Fanuc TP program (LS listing): layer_407.ls

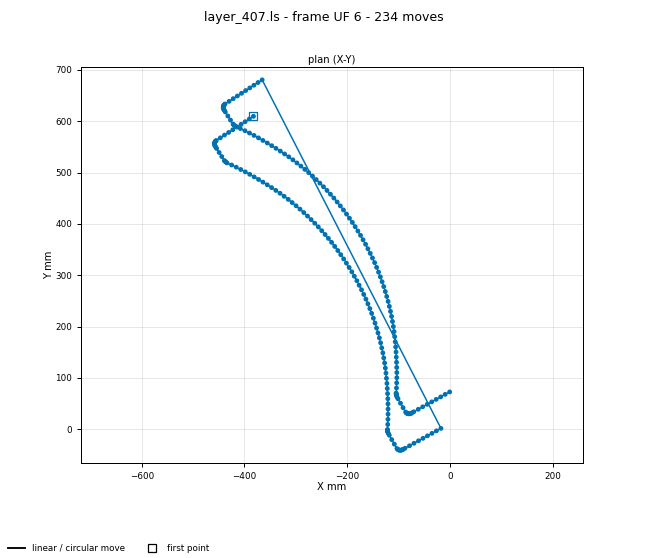
[picture p0: tool path of layer_407.ls in frame UF 6, 234 of 234 moves have a stored position in this frame; points joined in program order, loops and branches not executed]
/PROG layer_407
/ATTR
OWNER       = MNEDITOR;
CREATE      = DATE 100-11-20  TIME 09:43:21;
MODIFIED    = DATE 100-12-05  TIME 05:26:29;
LINE_COUNT = 119;
PROTECT     = READ_WRITE;
TCD:  STACK_SIZE    = 0,
      TASK_PRIORITY = 50,
      TIME_SLICE    = 0,
      BUSY_LAMP_OFF = 0,
      ABORT_REQUEST = 0,
      PAUSE_REQUEST = 0;
DEFAULT_GROUP   = 1,1,*,*,*;
CONTROL_CODE    = 00000000 00000000;
/MN
:R[35]=920.0;
:R[34]=0;
1: L P[1] 240cm/min CNT100 COORD ;
: Arc Start[1];
2: L P[2] 240cm/min CNT100 COORD PTH ;
3: L P[3] 240cm/min CNT100 COORD PTH ;
4: L P[4] 240cm/min CNT100 COORD PTH ;
5: L P[5] 240cm/min CNT100 COORD PTH ;
6: L P[6] 240cm/min CNT100 COORD PTH ;
7: L P[7] 240cm/min CNT100 COORD PTH ;
8: L P[8] 240cm/min CNT100 COORD PTH ;
9: L P[9] 240cm/min CNT100 COORD PTH ;
10: L P[10] 240cm/min CNT100 COORD PTH ;
11: L P[11] 240cm/min CNT100 COORD PTH ;
12: L P[12] 240cm/min CNT100 COORD PTH ;
13: L P[13] 240cm/min CNT100 COORD PTH ;
14: L P[14] 240cm/min CNT100 COORD PTH ;
15: L P[15] 240cm/min CNT100 COORD PTH ;
16: L P[16] 240cm/min CNT100 COORD PTH ;
17: L P[17] 240cm/min CNT100 COORD PTH ;
18: L P[18] 240cm/min CNT100 COORD PTH ;
19: L P[19] 240cm/min CNT100 COORD PTH ;
20: L P[20] 240cm/min CNT100 COORD PTH ;
21: L P[21] 240cm/min CNT100 COORD PTH ;
22: L P[22] 240cm/min CNT100 COORD PTH ;
23: L P[23] 240cm/min CNT100 COORD PTH ;
24: L P[24] 240cm/min CNT100 COORD PTH ;
25: L P[25] 240cm/min CNT100 COORD PTH ;
26: L P[26] 240cm/min CNT100 COORD PTH ;
27: L P[27] 240cm/min CNT100 COORD PTH ;
28: L P[28] 240cm/min CNT100 COORD PTH ;
29: L P[29] 240cm/min CNT100 COORD PTH ;
30: L P[30] 240cm/min CNT100 COORD PTH ;
31: L P[31] 240cm/min CNT100 COORD PTH ;
32: L P[32] 240cm/min CNT100 COORD PTH ;
33: L P[33] 240cm/min CNT100 COORD PTH ;
34: L P[34] 240cm/min CNT100 COORD PTH ;
35: L P[35] 240cm/min CNT100 COORD PTH ;
36: L P[36] 240cm/min CNT100 COORD PTH ;
37: L P[37] 240cm/min CNT100 COORD PTH ;
38: L P[38] 240cm/min CNT100 COORD PTH ;
39: L P[39] 240cm/min CNT100 COORD PTH ;
40: L P[40] 240cm/min CNT100 COORD PTH ;
41: L P[41] 240cm/min CNT100 COORD PTH ;
42: L P[42] 240cm/min CNT100 COORD PTH ;
43: L P[43] 240cm/min CNT100 COORD PTH ;
44: L P[44] 240cm/min CNT100 COORD PTH ;
45: L P[45] 240cm/min CNT100 COORD PTH ;
46: L P[46] 240cm/min CNT100 COORD PTH ;
47: L P[47] 240cm/min CNT100 COORD PTH ;
48: L P[48] 240cm/min CNT100 COORD PTH ;
49: L P[49] 240cm/min CNT100 COORD PTH ;
50: L P[50] 240cm/min CNT100 COORD PTH ;
51: L P[51] 240cm/min CNT100 COORD PTH ;
52: L P[52] 240cm/min CNT100 COORD PTH ;
53: L P[53] 240cm/min CNT100 COORD PTH ;
54: L P[54] 240cm/min CNT100 COORD PTH ;
55: L P[55] 240cm/min CNT100 COORD PTH ;
56: L P[56] 240cm/min CNT100 COORD PTH ;
57: L P[57] 240cm/min CNT100 COORD PTH ;
58: L P[58] 240cm/min CNT100 COORD PTH ;
59: L P[59] 240cm/min CNT100 COORD PTH ;
60: L P[60] 240cm/min CNT100 COORD PTH ;
61: L P[61] 240cm/min CNT100 COORD PTH ;
62: L P[62] 240cm/min CNT100 COORD PTH ;
63: L P[63] 240cm/min CNT100 COORD PTH ;
64: L P[64] 240cm/min CNT100 COORD PTH ;
65: L P[65] 240cm/min CNT100 COORD PTH ;
66: L P[66] 240cm/min CNT100 COORD PTH ;
67: L P[67] 240cm/min CNT100 COORD PTH ;
68: L P[68] 240cm/min CNT100 COORD PTH ;
69: L P[69] 240cm/min CNT100 COORD PTH ;
70: L P[70] 240cm/min CNT100 COORD PTH ;
71: L P[71] 240cm/min CNT100 COORD PTH ;
72: L P[72] 240cm/min CNT100 COORD PTH ;
73: L P[73] 240cm/min CNT100 COORD PTH ;
74: L P[74] 240cm/min CNT100 COORD PTH ;
75: L P[75] 240cm/min CNT100 COORD PTH ;
76: L P[76] 240cm/min CNT100 COORD PTH ;
77: L P[77] 240cm/min CNT100 COORD PTH ;
78: L P[78] 240cm/min CNT100 COORD PTH ;
79: L P[79] 240cm/min CNT100 COORD PTH ;
80: L P[80] 240cm/min CNT100 COORD PTH ;
81: L P[81] 240cm/min CNT100 COORD PTH ;
82: L P[82] 240cm/min CNT100 COORD PTH ;
83: L P[83] 240cm/min CNT100 COORD PTH ;
84: L P[84] 240cm/min CNT100 COORD PTH ;
85: L P[85] 240cm/min CNT100 COORD PTH ;
86: L P[86] 240cm/min CNT100 COORD PTH ;
87: L P[87] 240cm/min CNT100 COORD PTH ;
88: L P[88] 240cm/min CNT100 COORD PTH ;
89: L P[89] 240cm/min CNT100 COORD PTH ;
90: L P[90] 240cm/min CNT100 COORD PTH ;
91: L P[91] 240cm/min CNT100 COORD PTH ;
92: L P[92] 240cm/min CNT100 COORD PTH ;
93: L P[93] 240cm/min CNT100 COORD PTH ;
94: L P[94] 240cm/min CNT100 COORD PTH ;
95: L P[95] 240cm/min CNT100 COORD PTH ;
96: L P[96] 240cm/min CNT100 COORD PTH ;
97: L P[97] 240cm/min CNT100 COORD PTH ;
98: L P[98] 240cm/min CNT100 COORD PTH ;
99: L P[99] 240cm/min CNT100 COORD PTH ;
100: L P[100] 240cm/min CNT100 COORD PTH ;
101: L P[101] 240cm/min CNT100 COORD PTH ;
102: L P[102] 240cm/min CNT100 COORD PTH ;
103: L P[103] 240cm/min CNT100 COORD PTH ;
104: L P[104] 240cm/min CNT100 COORD PTH ;
105: L P[105] 240cm/min CNT100 COORD PTH ;
106: L P[106] 240cm/min CNT100 COORD PTH ;
107: L P[107] 240cm/min CNT100 COORD PTH ;
108: L P[108] 240cm/min CNT100 COORD PTH ;
109: L P[109] 240cm/min CNT100 COORD PTH ;
110: L P[110] 240cm/min CNT100 COORD PTH ;
111: L P[111] 240cm/min CNT100 COORD PTH ;
112: L P[112] 240cm/min CNT100 COORD PTH ;
113: L P[113] 240cm/min CNT100 COORD PTH ;
114: L P[114] 240cm/min CNT100 COORD PTH ;
115: L P[115] 240cm/min CNT100 COORD PTH ;
116: L P[116] 240cm/min CNT100 COORD PTH ;
117: L P[117] 240cm/min CNT100 COORD PTH ;
: Arc End[1];
:R[34]=1;
:SR[23]=$SCR_GRP[1].$MCH_POS_X;
:SR[24]=$SCR_GRP[1].$MCH_POS_Y;
120: L P[120] 800cm/min CNT100 COORD ;
:SR[23]=$SCR_GRP[1].$MCH_POS_X;
:SR[24]=$SCR_GRP[1].$MCH_POS_Y;
121: L P[121] 800cm/min CNT100 COORD PTH ;
:SR[23]=$SCR_GRP[1].$MCH_POS_X;
:SR[24]=$SCR_GRP[1].$MCH_POS_Y;
122: L P[122] 800cm/min CNT100 COORD PTH ;
:SR[23]=$SCR_GRP[1].$MCH_POS_X;
:SR[24]=$SCR_GRP[1].$MCH_POS_Y;
123: L P[123] 800cm/min CNT100 COORD PTH ;
:SR[23]=$SCR_GRP[1].$MCH_POS_X;
:SR[24]=$SCR_GRP[1].$MCH_POS_Y;
124: L P[124] 800cm/min CNT100 COORD PTH ;
:SR[23]=$SCR_GRP[1].$MCH_POS_X;
:SR[24]=$SCR_GRP[1].$MCH_POS_Y;
125: L P[125] 800cm/min CNT100 COORD PTH ;
:SR[23]=$SCR_GRP[1].$MCH_POS_X;
:SR[24]=$SCR_GRP[1].$MCH_POS_Y;
126: L P[126] 800cm/min CNT100 COORD PTH ;
:SR[23]=$SCR_GRP[1].$MCH_POS_X;
:SR[24]=$SCR_GRP[1].$MCH_POS_Y;
127: L P[127] 800cm/min CNT100 COORD PTH ;
:SR[23]=$SCR_GRP[1].$MCH_POS_X;
:SR[24]=$SCR_GRP[1].$MCH_POS_Y;
128: L P[128] 800cm/min CNT100 COORD PTH ;
:SR[23]=$SCR_GRP[1].$MCH_POS_X;
:SR[24]=$SCR_GRP[1].$MCH_POS_Y;
129: L P[129] 800cm/min CNT100 COORD PTH ;
:SR[23]=$SCR_GRP[1].$MCH_POS_X;
:SR[24]=$SCR_GRP[1].$MCH_POS_Y;
130: L P[130] 800cm/min CNT100 COORD PTH ;
:SR[23]=$SCR_GRP[1].$MCH_POS_X;
:SR[24]=$SCR_GRP[1].$MCH_POS_Y;
131: L P[131] 800cm/min CNT100 COORD PTH ;
:SR[23]=$SCR_GRP[1].$MCH_POS_X;
:SR[24]=$SCR_GRP[1].$MCH_POS_Y;
132: L P[132] 800cm/min CNT100 COORD PTH ;
:SR[23]=$SCR_GRP[1].$MCH_POS_X;
:SR[24]=$SCR_GRP[1].$MCH_POS_Y;
133: L P[133] 800cm/min CNT100 COORD PTH ;
:SR[23]=$SCR_GRP[1].$MCH_POS_X;
:SR[24]=$SCR_GRP[1].$MCH_POS_Y;
134: L P[134] 800cm/min CNT100 COORD PTH ;
:SR[23]=$SCR_GRP[1].$MCH_POS_X;
:SR[24]=$SCR_GRP[1].$MCH_POS_Y;
135: L P[135] 800cm/min CNT100 COORD PTH ;
:SR[23]=$SCR_GRP[1].$MCH_POS_X;
:SR[24]=$SCR_GRP[1].$MCH_POS_Y;
136: L P[136] 800cm/min CNT100 COORD PTH ;
:SR[23]=$SCR_GRP[1].$MCH_POS_X;
:SR[24]=$SCR_GRP[1].$MCH_POS_Y;
137: L P[137] 800cm/min CNT100 COORD PTH ;
:SR[23]=$SCR_GRP[1].$MCH_POS_X;
:SR[24]=$SCR_GRP[1].$MCH_POS_Y;
138: L P[138] 800cm/min CNT100 COORD PTH ;
:SR[23]=$SCR_GRP[1].$MCH_POS_X;
:SR[24]=$SCR_GRP[1].$MCH_POS_Y;
139: L P[139] 800cm/min CNT100 COORD PTH ;
:SR[23]=$SCR_GRP[1].$MCH_POS_X;
:SR[24]=$SCR_GRP[1].$MCH_POS_Y;
140: L P[140] 800cm/min CNT100 COORD PTH ;
:SR[23]=$SCR_GRP[1].$MCH_POS_X;
:SR[24]=$SCR_GRP[1].$MCH_POS_Y;
141: L P[141] 800cm/min CNT100 COORD PTH ;
:SR[23]=$SCR_GRP[1].$MCH_POS_X;
:SR[24]=$SCR_GRP[1].$MCH_POS_Y;
142: L P[142] 800cm/min CNT100 COORD PTH ;
:SR[23]=$SCR_GRP[1].$MCH_POS_X;
:SR[24]=$SCR_GRP[1].$MCH_POS_Y;
143: L P[143] 800cm/min CNT100 COORD PTH ;
:SR[23]=$SCR_GRP[1].$MCH_POS_X;
:SR[24]=$SCR_GRP[1].$MCH_POS_Y;
144: L P[144] 800cm/min CNT100 COORD PTH ;
:SR[23]=$SCR_GRP[1].$MCH_POS_X;
:SR[24]=$SCR_GRP[1].$MCH_POS_Y;
145: L P[145] 800cm/min CNT100 COORD PTH ;
:SR[23]=$SCR_GRP[1].$MCH_POS_X;
:SR[24]=$SCR_GRP[1].$MCH_POS_Y;
146: L P[146] 800cm/min CNT100 COORD PTH ;
:SR[23]=$SCR_GRP[1].$MCH_POS_X;
:SR[24]=$SCR_GRP[1].$MCH_POS_Y;
147: L P[147] 800cm/min CNT100 COORD PTH ;
:SR[23]=$SCR_GRP[1].$MCH_POS_X;
:SR[24]=$SCR_GRP[1].$MCH_POS_Y;
148: L P[148] 800cm/min CNT100 COORD PTH ;
:SR[23]=$SCR_GRP[1].$MCH_POS_X;
:SR[24]=$SCR_GRP[1].$MCH_POS_Y;
149: L P[149] 800cm/min CNT100 COORD PTH ;
:SR[23]=$SCR_GRP[1].$MCH_POS_X;
:SR[24]=$SCR_GRP[1].$MCH_POS_Y;
150: L P[150] 800cm/min CNT100 COORD PTH ;
:SR[23]=$SCR_GRP[1].$MCH_POS_X;
:SR[24]=$SCR_GRP[1].$MCH_POS_Y;
151: L P[151] 800cm/min CNT100 COORD PTH ;
:SR[23]=$SCR_GRP[1].$MCH_POS_X;
:SR[24]=$SCR_GRP[1].$MCH_POS_Y;
152: L P[152] 800cm/min CNT100 COORD PTH ;
:SR[23]=$SCR_GRP[1].$MCH_POS_X;
:SR[24]=$SCR_GRP[1].$MCH_POS_Y;
153: L P[153] 800cm/min CNT100 COORD PTH ;
:SR[23]=$SCR_GRP[1].$MCH_POS_X;
:SR[24]=$SCR_GRP[1].$MCH_POS_Y;
154: L P[154] 800cm/min CNT100 COORD PTH ;
:SR[23]=$SCR_GRP[1].$MCH_POS_X;
:SR[24]=$SCR_GRP[1].$MCH_POS_Y;
155: L P[155] 800cm/min CNT100 COORD PTH ;
:SR[23]=$SCR_GRP[1].$MCH_POS_X;
:SR[24]=$SCR_GRP[1].$MCH_POS_Y;
156: L P[156] 800cm/min CNT100 COORD PTH ;
:SR[23]=$SCR_GRP[1].$MCH_POS_X;
:SR[24]=$SCR_GRP[1].$MCH_POS_Y;
157: L P[157] 800cm/min CNT100 COORD PTH ;
:SR[23]=$SCR_GRP[1].$MCH_POS_X;
:SR[24]=$SCR_GRP[1].$MCH_POS_Y;
158: L P[158] 800cm/min CNT100 COORD PTH ;
:SR[23]=$SCR_GRP[1].$MCH_POS_X;
:SR[24]=$SCR_GRP[1].$MCH_POS_Y;
159: L P[159] 800cm/min CNT100 COORD PTH ;
:SR[23]=$SCR_GRP[1].$MCH_POS_X;
:SR[24]=$SCR_GRP[1].$MCH_POS_Y;
160: L P[160] 800cm/min CNT100 COORD PTH ;
:SR[23]=$SCR_GRP[1].$MCH_POS_X;
:SR[24]=$SCR_GRP[1].$MCH_POS_Y;
161: L P[161] 800cm/min CNT100 COORD PTH ;
:SR[23]=$SCR_GRP[1].$MCH_POS_X;
:SR[24]=$SCR_GRP[1].$MCH_POS_Y;
162: L P[162] 800cm/min CNT100 COORD PTH ;
:SR[23]=$SCR_GRP[1].$MCH_POS_X;
:SR[24]=$SCR_GRP[1].$MCH_POS_Y;
163: L P[163] 800cm/min CNT100 COORD PTH ;
:SR[23]=$SCR_GRP[1].$MCH_POS_X;
:SR[24]=$SCR_GRP[1].$MCH_POS_Y;
164: L P[164] 800cm/min CNT100 COORD PTH ;
:SR[23]=$SCR_GRP[1].$MCH_POS_X;
:SR[24]=$SCR_GRP[1].$MCH_POS_Y;
165: L P[165] 800cm/min CNT100 COORD PTH ;
:SR[23]=$SCR_GRP[1].$MCH_POS_X;
:SR[24]=$SCR_GRP[1].$MCH_POS_Y;
166: L P[166] 800cm/min CNT100 COORD PTH ;
:SR[23]=$SCR_GRP[1].$MCH_POS_X;
:SR[24]=$SCR_GRP[1].$MCH_POS_Y;
167: L P[167] 800cm/min CNT100 COORD PTH ;
:SR[23]=$SCR_GRP[1].$MCH_POS_X;
:SR[24]=$SCR_GRP[1].$MCH_POS_Y;
168: L P[168] 800cm/min CNT100 COORD PTH ;
:SR[23]=$SCR_GRP[1].$MCH_POS_X;
:SR[24]=$SCR_GRP[1].$MCH_POS_Y;
169: L P[169] 800cm/min CNT100 COORD PTH ;
:SR[23]=$SCR_GRP[1].$MCH_POS_X;
:SR[24]=$SCR_GRP[1].$MCH_POS_Y;
170: L P[170] 800cm/min CNT100 COORD PTH ;
:SR[23]=$SCR_GRP[1].$MCH_POS_X;
:SR[24]=$SCR_GRP[1].$MCH_POS_Y;
171: L P[171] 800cm/min CNT100 COORD PTH ;
:SR[23]=$SCR_GRP[1].$MCH_POS_X;
:SR[24]=$SCR_GRP[1].$MCH_POS_Y;
172: L P[172] 800cm/min CNT100 COORD PTH ;
:SR[23]=$SCR_GRP[1].$MCH_POS_X;
:SR[24]=$SCR_GRP[1].$MCH_POS_Y;
173: L P[173] 800cm/min CNT100 COORD PTH ;
:SR[23]=$SCR_GRP[1].$MCH_POS_X;
:SR[24]=$SCR_GRP[1].$MCH_POS_Y;
174: L P[174] 800cm/min CNT100 COORD PTH ;
:SR[23]=$SCR_GRP[1].$MCH_POS_X;
:SR[24]=$SCR_GRP[1].$MCH_POS_Y;
175: L P[175] 800cm/min CNT100 COORD PTH ;
:SR[23]=$SCR_GRP[1].$MCH_POS_X;
:SR[24]=$SCR_GRP[1].$MCH_POS_Y;
176: L P[176] 800cm/min CNT100 COORD PTH ;
:SR[23]=$SCR_GRP[1].$MCH_POS_X;
:SR[24]=$SCR_GRP[1].$MCH_POS_Y;
177: L P[177] 800cm/min CNT100 COORD PTH ;
:SR[23]=$SCR_GRP[1].$MCH_POS_X;
:SR[24]=$SCR_GRP[1].$MCH_POS_Y;
178: L P[178] 800cm/min CNT100 COORD PTH ;
:SR[23]=$SCR_GRP[1].$MCH_POS_X;
:SR[24]=$SCR_GRP[1].$MCH_POS_Y;
179: L P[179] 800cm/min CNT100 COORD PTH ;
:SR[23]=$SCR_GRP[1].$MCH_POS_X;
:SR[24]=$SCR_GRP[1].$MCH_POS_Y;
180: L P[180] 800cm/min CNT100 COORD PTH ;
:SR[23]=$SCR_GRP[1].$MCH_POS_X;
:SR[24]=$SCR_GRP[1].$MCH_POS_Y;
181: L P[181] 800cm/min CNT100 COORD PTH ;
:SR[23]=$SCR_GRP[1].$MCH_POS_X;
:SR[24]=$SCR_GRP[1].$MCH_POS_Y;
182: L P[182] 800cm/min CNT100 COORD PTH ;
:SR[23]=$SCR_GRP[1].$MCH_POS_X;
:SR[24]=$SCR_GRP[1].$MCH_POS_Y;
183: L P[183] 800cm/min CNT100 COORD PTH ;
:SR[23]=$SCR_GRP[1].$MCH_POS_X;
:SR[24]=$SCR_GRP[1].$MCH_POS_Y;
184: L P[184] 800cm/min CNT100 COORD PTH ;
:SR[23]=$SCR_GRP[1].$MCH_POS_X;
:SR[24]=$SCR_GRP[1].$MCH_POS_Y;
185: L P[185] 800cm/min CNT100 COORD PTH ;
:SR[23]=$SCR_GRP[1].$MCH_POS_X;
:SR[24]=$SCR_GRP[1].$MCH_POS_Y;
186: L P[186] 800cm/min CNT100 COORD PTH ;
:SR[23]=$SCR_GRP[1].$MCH_POS_X;
:SR[24]=$SCR_GRP[1].$MCH_POS_Y;
187: L P[187] 800cm/min CNT100 COORD PTH ;
:SR[23]=$SCR_GRP[1].$MCH_POS_X;
:SR[24]=$SCR_GRP[1].$MCH_POS_Y;
188: L P[188] 800cm/min CNT100 COORD PTH ;
:SR[23]=$SCR_GRP[1].$MCH_POS_X;
:SR[24]=$SCR_GRP[1].$MCH_POS_Y;
189: L P[189] 800cm/min CNT100 COORD PTH ;
:SR[23]=$SCR_GRP[1].$MCH_POS_X;
:SR[24]=$SCR_GRP[1].$MCH_POS_Y;
190: L P[190] 800cm/min CNT100 COORD PTH ;
:SR[23]=$SCR_GRP[1].$MCH_POS_X;
:SR[24]=$SCR_GRP[1].$MCH_POS_Y;
191: L P[191] 800cm/min CNT100 COORD PTH ;
:SR[23]=$SCR_GRP[1].$MCH_POS_X;
:SR[24]=$SCR_GRP[1].$MCH_POS_Y;
192: L P[192] 800cm/min CNT100 COORD PTH ;
:SR[23]=$SCR_GRP[1].$MCH_POS_X;
:SR[24]=$SCR_GRP[1].$MCH_POS_Y;
193: L P[193] 800cm/min CNT100 COORD PTH ;
:SR[23]=$SCR_GRP[1].$MCH_POS_X;
:SR[24]=$SCR_GRP[1].$MCH_POS_Y;
194: L P[194] 800cm/min CNT100 COORD PTH ;
:SR[23]=$SCR_GRP[1].$MCH_POS_X;
:SR[24]=$SCR_GRP[1].$MCH_POS_Y;
195: L P[195] 800cm/min CNT100 COORD PTH ;
:SR[23]=$SCR_GRP[1].$MCH_POS_X;
:SR[24]=$SCR_GRP[1].$MCH_POS_Y;
196: L P[196] 800cm/min CNT100 COORD PTH ;
:SR[23]=$SCR_GRP[1].$MCH_POS_X;
:SR[24]=$SCR_GRP[1].$MCH_POS_Y;
197: L P[197] 800cm/min CNT100 COORD PTH ;
:SR[23]=$SCR_GRP[1].$MCH_POS_X;
:SR[24]=$SCR_GRP[1].$MCH_POS_Y;
198: L P[198] 800cm/min CNT100 COORD PTH ;
:SR[23]=$SCR_GRP[1].$MCH_POS_X;
:SR[24]=$SCR_GRP[1].$MCH_POS_Y;
199: L P[199] 800cm/min CNT100 COORD PTH ;
:SR[23]=$SCR_GRP[1].$MCH_POS_X;
:SR[24]=$SCR_GRP[1].$MCH_POS_Y;
200: L P[200] 800cm/min CNT100 COORD PTH ;
:SR[23]=$SCR_GRP[1].$MCH_POS_X;
:SR[24]=$SCR_GRP[1].$MCH_POS_Y;
201: L P[201] 800cm/min CNT100 COORD PTH ;
:SR[23]=$SCR_GRP[1].$MCH_POS_X;
:SR[24]=$SCR_GRP[1].$MCH_POS_Y;
202: L P[202] 800cm/min CNT100 COORD PTH ;
:SR[23]=$SCR_GRP[1].$MCH_POS_X;
:SR[24]=$SCR_GRP[1].$MCH_POS_Y;
203: L P[203] 800cm/min CNT100 COORD PTH ;
:SR[23]=$SCR_GRP[1].$MCH_POS_X;
:SR[24]=$SCR_GRP[1].$MCH_POS_Y;
204: L P[204] 800cm/min CNT100 COORD PTH ;
:SR[23]=$SCR_GRP[1].$MCH_POS_X;
:SR[24]=$SCR_GRP[1].$MCH_POS_Y;
205: L P[205] 800cm/min CNT100 COORD PTH ;
:SR[23]=$SCR_GRP[1].$MCH_POS_X;
:SR[24]=$SCR_GRP[1].$MCH_POS_Y;
206: L P[206] 800cm/min CNT100 COORD PTH ;
:SR[23]=$SCR_GRP[1].$MCH_POS_X;
:SR[24]=$SCR_GRP[1].$MCH_POS_Y;
207: L P[207] 800cm/min CNT100 COORD PTH ;
:SR[23]=$SCR_GRP[1].$MCH_POS_X;
:SR[24]=$SCR_GRP[1].$MCH_POS_Y;
208: L P[208] 800cm/min CNT100 COORD PTH ;
:SR[23]=$SCR_GRP[1].$MCH_POS_X;
:SR[24]=$SCR_GRP[1].$MCH_POS_Y;
209: L P[209] 800cm/min CNT100 COORD PTH ;
:SR[23]=$SCR_GRP[1].$MCH_POS_X;
:SR[24]=$SCR_GRP[1].$MCH_POS_Y;
210: L P[210] 800cm/min CNT100 COORD PTH ;
:SR[23]=$SCR_GRP[1].$MCH_POS_X;
:SR[24]=$SCR_GRP[1].$MCH_POS_Y;
211: L P[211] 800cm/min CNT100 COORD PTH ;
:SR[23]=$SCR_GRP[1].$MCH_POS_X;
:SR[24]=$SCR_GRP[1].$MCH_POS_Y;
212: L P[212] 800cm/min CNT100 COORD PTH ;
:SR[23]=$SCR_GRP[1].$MCH_POS_X;
:SR[24]=$SCR_GRP[1].$MCH_POS_Y;
213: L P[213] 800cm/min CNT100 COORD PTH ;
:SR[23]=$SCR_GRP[1].$MCH_POS_X;
:SR[24]=$SCR_GRP[1].$MCH_POS_Y;
214: L P[214] 800cm/min CNT100 COORD PTH ;
:SR[23]=$SCR_GRP[1].$MCH_POS_X;
:SR[24]=$SCR_GRP[1].$MCH_POS_Y;
215: L P[215] 800cm/min CNT100 COORD PTH ;
:SR[23]=$SCR_GRP[1].$MCH_POS_X;
:SR[24]=$SCR_GRP[1].$MCH_POS_Y;
216: L P[216] 800cm/min CNT100 COORD PTH ;
:SR[23]=$SCR_GRP[1].$MCH_POS_X;
:SR[24]=$SCR_GRP[1].$MCH_POS_Y;
217: L P[217] 800cm/min CNT100 COORD PTH ;
:SR[23]=$SCR_GRP[1].$MCH_POS_X;
:SR[24]=$SCR_GRP[1].$MCH_POS_Y;
218: L P[218] 800cm/min CNT100 COORD PTH ;
:SR[23]=$SCR_GRP[1].$MCH_POS_X;
:SR[24]=$SCR_GRP[1].$MCH_POS_Y;
219: L P[219] 800cm/min CNT100 COORD PTH ;
:SR[23]=$SCR_GRP[1].$MCH_POS_X;
:SR[24]=$SCR_GRP[1].$MCH_POS_Y;
220: L P[220] 800cm/min CNT100 COORD PTH ;
:SR[23]=$SCR_GRP[1].$MCH_POS_X;
:SR[24]=$SCR_GRP[1].$MCH_POS_Y;
221: L P[221] 800cm/min CNT100 COORD PTH ;
:SR[23]=$SCR_GRP[1].$MCH_POS_X;
:SR[24]=$SCR_GRP[1].$MCH_POS_Y;
222: L P[222] 800cm/min CNT100 COORD PTH ;
:SR[23]=$SCR_GRP[1].$MCH_POS_X;
:SR[24]=$SCR_GRP[1].$MCH_POS_Y;
223: L P[223] 800cm/min CNT100 COORD PTH ;
:SR[23]=$SCR_GRP[1].$MCH_POS_X;
:SR[24]=$SCR_GRP[1].$MCH_POS_Y;
224: L P[224] 800cm/min CNT100 COORD PTH ;
:SR[23]=$SCR_GRP[1].$MCH_POS_X;
:SR[24]=$SCR_GRP[1].$MCH_POS_Y;
225: L P[225] 800cm/min CNT100 COORD PTH ;
:SR[23]=$SCR_GRP[1].$MCH_POS_X;
:SR[24]=$SCR_GRP[1].$MCH_POS_Y;
226: L P[226] 800cm/min CNT100 COORD PTH ;
:SR[23]=$SCR_GRP[1].$MCH_POS_X;
:SR[24]=$SCR_GRP[1].$MCH_POS_Y;
227: L P[227] 800cm/min CNT100 COORD PTH ;
:SR[23]=$SCR_GRP[1].$MCH_POS_X;
:SR[24]=$SCR_GRP[1].$MCH_POS_Y;
228: L P[228] 800cm/min CNT100 COORD PTH ;
:SR[23]=$SCR_GRP[1].$MCH_POS_X;
:SR[24]=$SCR_GRP[1].$MCH_POS_Y;
229: L P[229] 800cm/min CNT100 COORD PTH ;
:SR[23]=$SCR_GRP[1].$MCH_POS_X;
:SR[24]=$SCR_GRP[1].$MCH_POS_Y;
230: L P[230] 800cm/min CNT100 COORD PTH ;
:SR[23]=$SCR_GRP[1].$MCH_POS_X;
:SR[24]=$SCR_GRP[1].$MCH_POS_Y;
231: L P[231] 800cm/min CNT100 COORD PTH ;
:SR[23]=$SCR_GRP[1].$MCH_POS_X;
:SR[24]=$SCR_GRP[1].$MCH_POS_Y;
232: L P[232] 800cm/min CNT100 COORD PTH ;
:SR[23]=$SCR_GRP[1].$MCH_POS_X;
:SR[24]=$SCR_GRP[1].$MCH_POS_Y;
233: L P[233] 800cm/min CNT100 COORD PTH ;
:SR[23]=$SCR_GRP[1].$MCH_POS_X;
:SR[24]=$SCR_GRP[1].$MCH_POS_Y;
234: L P[234] 800cm/min CNT100 COORD PTH ;
:SR[23]=$SCR_GRP[1].$MCH_POS_X;
:SR[24]=$SCR_GRP[1].$MCH_POS_Y;
235: L P[235] 800cm/min CNT100 COORD PTH ;
:SR[23]=$SCR_GRP[1].$MCH_POS_X;
:SR[24]=$SCR_GRP[1].$MCH_POS_Y;
236: L P[236] 800cm/min CNT100 COORD PTH ;
:R[34]=0;
/POS
P[1] {
    GP1:
        UF : 6, UT : 5,     CONFIG: 'N U T, 0, 0, 0',
       X = -382.5 mm, Y = 609.6 mm, Z = 920.0 mm,
       W = 0.0 deg, P = 0.0 deg,
    GP2:
        UF : 1, UT : 2,
       J1 = 0.0 deg, J2 = 0.0 deg
 };
P[120] {
    GP1:
        UF : 6, UT : 5,     CONFIG: 'N U T, 0, 0, 0',
 X = -365.5 mm, Y = 680.6 mm, Z = 920.0 mm,       W = 0.0 deg, P = 0.0 deg,
    GP2:
        UF : 1, UT : 2,
       J1 = 0.0 deg, J2 = 0.0 deg
 };
P[2] {
    GP1:
        UF : 6, UT : 5,     CONFIG: 'N U T, 0, 0, 0',
       X = -390.5 mm, Y = 604.4 mm, Z = 920.0 mm,
       W = 0.0 deg, P = 0.0 deg,
    GP2:
        UF : 1, UT : 2,
       J1 = 0.0 deg, J2 = 0.0 deg
 };
P[121] {
    GP1:
        UF : 6, UT : 5,     CONFIG: 'N U T, 0, 0, 0',
 X = -373.5 mm, Y = 675.4 mm, Z = 920.0 mm,       W = 0.0 deg, P = 0.0 deg,
    GP2:
        UF : 1, UT : 2,
       J1 = 0.0 deg, J2 = 0.0 deg
 };
P[3] {
    GP1:
        UF : 6, UT : 5,     CONFIG: 'N U T, 0, 0, 0',
       X = -398.6 mm, Y = 599.1 mm, Z = 920.0 mm,
       W = 0.0 deg, P = 0.0 deg,
    GP2:
        UF : 1, UT : 2,
       J1 = 0.0 deg, J2 = 0.0 deg
 };
P[122] {
    GP1:
        UF : 6, UT : 5,     CONFIG: 'N U T, 0, 0, 0',
 X = -381.6 mm, Y = 670.1 mm, Z = 920.0 mm,       W = 0.0 deg, P = 0.0 deg,
    GP2:
        UF : 1, UT : 2,
       J1 = 0.0 deg, J2 = 0.0 deg
 };
P[4] {
    GP1:
        UF : 6, UT : 5,     CONFIG: 'N U T, 0, 0, 0',
       X = -406.6 mm, Y = 593.9 mm, Z = 920.0 mm,
       W = 0.0 deg, P = 0.0 deg,
    GP2:
        UF : 1, UT : 2,
       J1 = 0.0 deg, J2 = 0.0 deg
 };
P[123] {
    GP1:
        UF : 6, UT : 5,     CONFIG: 'N U T, 0, 0, 0',
 X = -389.6 mm, Y = 664.9 mm, Z = 920.0 mm,       W = 0.0 deg, P = 0.0 deg,
    GP2:
        UF : 1, UT : 2,
       J1 = 0.0 deg, J2 = 0.0 deg
 };
P[5] {
    GP1:
        UF : 6, UT : 5,     CONFIG: 'N U T, 0, 0, 0',
       X = -414.7 mm, Y = 588.7 mm, Z = 920.0 mm,
       W = 0.0 deg, P = 0.0 deg,
    GP2:
        UF : 1, UT : 2,
       J1 = 0.0 deg, J2 = 0.0 deg
 };
P[124] {
    GP1:
        UF : 6, UT : 5,     CONFIG: 'N U T, 0, 0, 0',
 X = -397.7 mm, Y = 659.7 mm, Z = 920.0 mm,       W = 0.0 deg, P = 0.0 deg,
    GP2:
        UF : 1, UT : 2,
       J1 = 0.0 deg, J2 = 0.0 deg
 };
P[6] {
    GP1:
        UF : 6, UT : 5,     CONFIG: 'N U T, 0, 0, 0',
       X = -422.7 mm, Y = 583.4 mm, Z = 920.0 mm,
       W = 0.0 deg, P = 0.0 deg,
    GP2:
        UF : 1, UT : 2,
       J1 = 0.0 deg, J2 = 0.0 deg
 };
P[125] {
    GP1:
        UF : 6, UT : 5,     CONFIG: 'N U T, 0, 0, 0',
 X = -405.7 mm, Y = 654.4 mm, Z = 920.0 mm,       W = 0.0 deg, P = 0.0 deg,
    GP2:
        UF : 1, UT : 2,
       J1 = 0.0 deg, J2 = 0.0 deg
 };
P[7] {
    GP1:
        UF : 6, UT : 5,     CONFIG: 'N U T, 0, 0, 0',
       X = -430.8 mm, Y = 578.2 mm, Z = 920.0 mm,
       W = 0.0 deg, P = 0.0 deg,
    GP2:
        UF : 1, UT : 2,
       J1 = 0.0 deg, J2 = 0.0 deg
 };
P[126] {
    GP1:
        UF : 6, UT : 5,     CONFIG: 'N U T, 0, 0, 0',
 X = -413.8 mm, Y = 649.2 mm, Z = 920.0 mm,       W = 0.0 deg, P = 0.0 deg,
    GP2:
        UF : 1, UT : 2,
       J1 = 0.0 deg, J2 = 0.0 deg
 };
P[8] {
    GP1:
        UF : 6, UT : 5,     CONFIG: 'N U T, 0, 0, 0',
       X = -438.9 mm, Y = 573.0 mm, Z = 920.0 mm,
       W = 0.0 deg, P = 0.0 deg,
    GP2:
        UF : 1, UT : 2,
       J1 = 0.0 deg, J2 = 0.0 deg
 };
P[127] {
    GP1:
        UF : 6, UT : 5,     CONFIG: 'N U T, 0, 0, 0',
 X = -421.9 mm, Y = 644.0 mm, Z = 920.0 mm,       W = 0.0 deg, P = 0.0 deg,
    GP2:
        UF : 1, UT : 2,
       J1 = 0.0 deg, J2 = 0.0 deg
 };
P[9] {
    GP1:
        UF : 6, UT : 5,     CONFIG: 'N U T, 0, 0, 0',
       X = -446.9 mm, Y = 567.7 mm, Z = 920.0 mm,
       W = 0.0 deg, P = 0.0 deg,
    GP2:
        UF : 1, UT : 2,
       J1 = 0.0 deg, J2 = 0.0 deg
 };
P[128] {
    GP1:
        UF : 6, UT : 5,     CONFIG: 'N U T, 0, 0, 0',
 X = -429.9 mm, Y = 638.7 mm, Z = 920.0 mm,       W = 0.0 deg, P = 0.0 deg,
    GP2:
        UF : 1, UT : 2,
       J1 = 0.0 deg, J2 = 0.0 deg
 };
P[10] {
    GP1:
        UF : 6, UT : 5,     CONFIG: 'N U T, 0, 0, 0',
       X = -455.0 mm, Y = 562.5 mm, Z = 920.0 mm,
       W = 0.0 deg, P = 0.0 deg,
    GP2:
        UF : 1, UT : 2,
       J1 = 0.0 deg, J2 = 0.0 deg
 };
P[129] {
    GP1:
        UF : 6, UT : 5,     CONFIG: 'N U T, 0, 0, 0',
 X = -438.0 mm, Y = 633.5 mm, Z = 920.0 mm,       W = 0.0 deg, P = 0.0 deg,
    GP2:
        UF : 1, UT : 2,
       J1 = 0.0 deg, J2 = 0.0 deg
 };
P[11] {
    GP1:
        UF : 6, UT : 5,     CONFIG: 'N U T, 0, 0, 0',
       X = -456.0 mm, Y = 561.5 mm, Z = 920.0 mm,
       W = 0.0 deg, P = 0.0 deg,
    GP2:
        UF : 1, UT : 2,
       J1 = 0.0 deg, J2 = 0.0 deg
 };
P[130] {
    GP1:
        UF : 6, UT : 5,     CONFIG: 'N U T, 0, 0, 0',
 X = -439.0 mm, Y = 632.5 mm, Z = 920.0 mm,       W = 0.0 deg, P = 0.0 deg,
    GP2:
        UF : 1, UT : 2,
       J1 = 0.0 deg, J2 = 0.0 deg
 };
P[12] {
    GP1:
        UF : 6, UT : 5,     CONFIG: 'N U T, 0, 0, 0',
       X = -456.9 mm, Y = 560.5 mm, Z = 920.0 mm,
       W = 0.0 deg, P = 0.0 deg,
    GP2:
        UF : 1, UT : 2,
       J1 = 0.0 deg, J2 = 0.0 deg
 };
P[131] {
    GP1:
        UF : 6, UT : 5,     CONFIG: 'N U T, 0, 0, 0',
 X = -439.9 mm, Y = 631.5 mm, Z = 920.0 mm,       W = 0.0 deg, P = 0.0 deg,
    GP2:
        UF : 1, UT : 2,
       J1 = 0.0 deg, J2 = 0.0 deg
 };
P[13] {
    GP1:
        UF : 6, UT : 5,     CONFIG: 'N U T, 0, 0, 0',
       X = -457.5 mm, Y = 559.4 mm, Z = 920.0 mm,
       W = 0.0 deg, P = 0.0 deg,
    GP2:
        UF : 1, UT : 2,
       J1 = 0.0 deg, J2 = 0.0 deg
 };
P[132] {
    GP1:
        UF : 6, UT : 5,     CONFIG: 'N U T, 0, 0, 0',
 X = -440.5 mm, Y = 630.4 mm, Z = 920.0 mm,       W = 0.0 deg, P = 0.0 deg,
    GP2:
        UF : 1, UT : 2,
       J1 = 0.0 deg, J2 = 0.0 deg
 };
P[14] {
    GP1:
        UF : 6, UT : 5,     CONFIG: 'N U T, 0, 0, 0',
       X = -458.0 mm, Y = 558.1 mm, Z = 920.0 mm,
       W = 0.0 deg, P = 0.0 deg,
    GP2:
        UF : 1, UT : 2,
       J1 = 0.0 deg, J2 = 0.0 deg
 };
P[133] {
    GP1:
        UF : 6, UT : 5,     CONFIG: 'N U T, 0, 0, 0',
 X = -441.0 mm, Y = 629.1 mm, Z = 920.0 mm,       W = 0.0 deg, P = 0.0 deg,
    GP2:
        UF : 1, UT : 2,
       J1 = 0.0 deg, J2 = 0.0 deg
 };
P[15] {
    GP1:
        UF : 6, UT : 5,     CONFIG: 'N U T, 0, 0, 0',
       X = -458.3 mm, Y = 556.8 mm, Z = 920.0 mm,
       W = 0.0 deg, P = 0.0 deg,
    GP2:
        UF : 1, UT : 2,
       J1 = 0.0 deg, J2 = 0.0 deg
 };
P[134] {
    GP1:
        UF : 6, UT : 5,     CONFIG: 'N U T, 0, 0, 0',
 X = -441.3 mm, Y = 627.8 mm, Z = 920.0 mm,       W = 0.0 deg, P = 0.0 deg,
    GP2:
        UF : 1, UT : 2,
       J1 = 0.0 deg, J2 = 0.0 deg
 };
P[16] {
    GP1:
        UF : 6, UT : 5,     CONFIG: 'N U T, 0, 0, 0',
       X = -458.3 mm, Y = 555.2 mm, Z = 920.0 mm,
       W = 0.0 deg, P = 0.0 deg,
    GP2:
        UF : 1, UT : 2,
       J1 = 0.0 deg, J2 = 0.0 deg
 };
P[135] {
    GP1:
        UF : 6, UT : 5,     CONFIG: 'N U T, 0, 0, 0',
 X = -441.3 mm, Y = 626.2 mm, Z = 920.0 mm,       W = 0.0 deg, P = 0.0 deg,
    GP2:
        UF : 1, UT : 2,
       J1 = 0.0 deg, J2 = 0.0 deg
 };
P[17] {
    GP1:
        UF : 6, UT : 5,     CONFIG: 'N U T, 0, 0, 0',
       X = -457.9 mm, Y = 553.5 mm, Z = 920.0 mm,
       W = 0.0 deg, P = 0.0 deg,
    GP2:
        UF : 1, UT : 2,
       J1 = 0.0 deg, J2 = 0.0 deg
 };
P[136] {
    GP1:
        UF : 6, UT : 5,     CONFIG: 'N U T, 0, 0, 0',
 X = -440.9 mm, Y = 624.5 mm, Z = 920.0 mm,       W = 0.0 deg, P = 0.0 deg,
    GP2:
        UF : 1, UT : 2,
       J1 = 0.0 deg, J2 = 0.0 deg
 };
P[18] {
    GP1:
        UF : 6, UT : 5,     CONFIG: 'N U T, 0, 0, 0',
       X = -457.2 mm, Y = 551.9 mm, Z = 920.0 mm,
       W = 0.0 deg, P = 0.0 deg,
    GP2:
        UF : 1, UT : 2,
       J1 = 0.0 deg, J2 = 0.0 deg
 };
P[137] {
    GP1:
        UF : 6, UT : 5,     CONFIG: 'N U T, 0, 0, 0',
 X = -440.2 mm, Y = 622.9 mm, Z = 920.0 mm,       W = 0.0 deg, P = 0.0 deg,
    GP2:
        UF : 1, UT : 2,
       J1 = 0.0 deg, J2 = 0.0 deg
 };
P[19] {
    GP1:
        UF : 6, UT : 5,     CONFIG: 'N U T, 0, 0, 0',
       X = -455.8 mm, Y = 549.5 mm, Z = 920.0 mm,
       W = 0.0 deg, P = 0.0 deg,
    GP2:
        UF : 1, UT : 2,
       J1 = 0.0 deg, J2 = 0.0 deg
 };
P[138] {
    GP1:
        UF : 6, UT : 5,     CONFIG: 'N U T, 0, 0, 0',
 X = -438.8 mm, Y = 620.5 mm, Z = 920.0 mm,       W = 0.0 deg, P = 0.0 deg,
    GP2:
        UF : 1, UT : 2,
       J1 = 0.0 deg, J2 = 0.0 deg
 };
P[20] {
    GP1:
        UF : 6, UT : 5,     CONFIG: 'N U T, 0, 0, 0',
       X = -454.3 mm, Y = 547.1 mm, Z = 920.0 mm,
       W = 0.0 deg, P = 0.0 deg,
    GP2:
        UF : 1, UT : 2,
       J1 = 0.0 deg, J2 = 0.0 deg
 };
P[139] {
    GP1:
        UF : 6, UT : 5,     CONFIG: 'N U T, 0, 0, 0',
 X = -437.3 mm, Y = 618.1 mm, Z = 920.0 mm,       W = 0.0 deg, P = 0.0 deg,
    GP2:
        UF : 1, UT : 2,
       J1 = 0.0 deg, J2 = 0.0 deg
 };
P[21] {
    GP1:
        UF : 6, UT : 5,     CONFIG: 'N U T, 0, 0, 0',
       X = -449.3 mm, Y = 539.1 mm, Z = 920.0 mm,
       W = 0.0 deg, P = 0.0 deg,
    GP2:
        UF : 1, UT : 2,
       J1 = 0.0 deg, J2 = 0.0 deg
 };
P[140] {
    GP1:
        UF : 6, UT : 5,     CONFIG: 'N U T, 0, 0, 0',
 X = -432.3 mm, Y = 610.1 mm, Z = 920.0 mm,       W = 0.0 deg, P = 0.0 deg,
    GP2:
        UF : 1, UT : 2,
       J1 = 0.0 deg, J2 = 0.0 deg
 };
P[22] {
    GP1:
        UF : 6, UT : 5,     CONFIG: 'N U T, 0, 0, 0',
       X = -444.2 mm, Y = 531.2 mm, Z = 920.0 mm,
       W = 0.0 deg, P = 0.0 deg,
    GP2:
        UF : 1, UT : 2,
       J1 = 0.0 deg, J2 = 0.0 deg
 };
P[141] {
    GP1:
        UF : 6, UT : 5,     CONFIG: 'N U T, 0, 0, 0',
 X = -427.2 mm, Y = 602.2 mm, Z = 920.0 mm,       W = 0.0 deg, P = 0.0 deg,
    GP2:
        UF : 1, UT : 2,
       J1 = 0.0 deg, J2 = 0.0 deg
 };
P[23] {
    GP1:
        UF : 6, UT : 5,     CONFIG: 'N U T, 0, 0, 0',
       X = -439.1 mm, Y = 523.3 mm, Z = 920.0 mm,
       W = 0.0 deg, P = 0.0 deg,
    GP2:
        UF : 1, UT : 2,
       J1 = 0.0 deg, J2 = 0.0 deg
 };
P[142] {
    GP1:
        UF : 6, UT : 5,     CONFIG: 'N U T, 0, 0, 0',
 X = -422.1 mm, Y = 594.3 mm, Z = 920.0 mm,       W = 0.0 deg, P = 0.0 deg,
    GP2:
        UF : 1, UT : 2,
       J1 = 0.0 deg, J2 = 0.0 deg
 };
P[24] {
    GP1:
        UF : 6, UT : 5,     CONFIG: 'N U T, 0, 0, 0',
       X = -438.0 mm, Y = 522.1 mm, Z = 920.0 mm,
       W = 0.0 deg, P = 0.0 deg,
    GP2:
        UF : 1, UT : 2,
       J1 = 0.0 deg, J2 = 0.0 deg
 };
P[143] {
    GP1:
        UF : 6, UT : 5,     CONFIG: 'N U T, 0, 0, 0',
 X = -421.0 mm, Y = 593.1 mm, Z = 920.0 mm,       W = 0.0 deg, P = 0.0 deg,
    GP2:
        UF : 1, UT : 2,
       J1 = 0.0 deg, J2 = 0.0 deg
 };
P[25] {
    GP1:
        UF : 6, UT : 5,     CONFIG: 'N U T, 0, 0, 0',
       X = -435.8 mm, Y = 520.1 mm, Z = 920.0 mm,
       W = 0.0 deg, P = 0.0 deg,
    GP2:
        UF : 1, UT : 2,
       J1 = 0.0 deg, J2 = 0.0 deg
 };
P[144] {
    GP1:
        UF : 6, UT : 5,     CONFIG: 'N U T, 0, 0, 0',
 X = -418.8 mm, Y = 591.1 mm, Z = 920.0 mm,       W = 0.0 deg, P = 0.0 deg,
    GP2:
        UF : 1, UT : 2,
       J1 = 0.0 deg, J2 = 0.0 deg
 };
P[26] {
    GP1:
        UF : 6, UT : 5,     CONFIG: 'N U T, 0, 0, 0',
       X = -434.0 mm, Y = 518.9 mm, Z = 920.0 mm,
       W = 0.0 deg, P = 0.0 deg,
    GP2:
        UF : 1, UT : 2,
       J1 = 0.0 deg, J2 = 0.0 deg
 };
P[145] {
    GP1:
        UF : 6, UT : 5,     CONFIG: 'N U T, 0, 0, 0',
 X = -417.0 mm, Y = 589.9 mm, Z = 920.0 mm,       W = 0.0 deg, P = 0.0 deg,
    GP2:
        UF : 1, UT : 2,
       J1 = 0.0 deg, J2 = 0.0 deg
 };
P[27] {
    GP1:
        UF : 6, UT : 5,     CONFIG: 'N U T, 0, 0, 0',
       X = -425.0 mm, Y = 514.8 mm, Z = 920.0 mm,
       W = 0.0 deg, P = 0.0 deg,
    GP2:
        UF : 1, UT : 2,
       J1 = 0.0 deg, J2 = 0.0 deg
 };
P[146] {
    GP1:
        UF : 6, UT : 5,     CONFIG: 'N U T, 0, 0, 0',
 X = -408.0 mm, Y = 585.8 mm, Z = 920.0 mm,       W = 0.0 deg, P = 0.0 deg,
    GP2:
        UF : 1, UT : 2,
       J1 = 0.0 deg, J2 = 0.0 deg
 };
P[28] {
    GP1:
        UF : 6, UT : 5,     CONFIG: 'N U T, 0, 0, 0',
       X = -416.0 mm, Y = 510.5 mm, Z = 920.0 mm,
       W = 0.0 deg, P = 0.0 deg,
    GP2:
        UF : 1, UT : 2,
       J1 = 0.0 deg, J2 = 0.0 deg
 };
P[147] {
    GP1:
        UF : 6, UT : 5,     CONFIG: 'N U T, 0, 0, 0',
 X = -399.0 mm, Y = 581.5 mm, Z = 920.0 mm,       W = 0.0 deg, P = 0.0 deg,
    GP2:
        UF : 1, UT : 2,
       J1 = 0.0 deg, J2 = 0.0 deg
 };
P[29] {
    GP1:
        UF : 6, UT : 5,     CONFIG: 'N U T, 0, 0, 0',
       X = -407.2 mm, Y = 506.0 mm, Z = 920.0 mm,
       W = 0.0 deg, P = 0.0 deg,
    GP2:
        UF : 1, UT : 2,
       J1 = 0.0 deg, J2 = 0.0 deg
 };
P[148] {
    GP1:
        UF : 6, UT : 5,     CONFIG: 'N U T, 0, 0, 0',
 X = -390.2 mm, Y = 577.0 mm, Z = 920.0 mm,       W = 0.0 deg, P = 0.0 deg,
    GP2:
        UF : 1, UT : 2,
       J1 = 0.0 deg, J2 = 0.0 deg
 };
P[30] {
    GP1:
        UF : 6, UT : 5,     CONFIG: 'N U T, 0, 0, 0',
       X = -398.4 mm, Y = 501.4 mm, Z = 920.0 mm,
       W = 0.0 deg, P = 0.0 deg,
    GP2:
        UF : 1, UT : 2,
       J1 = 0.0 deg, J2 = 0.0 deg
 };
P[149] {
    GP1:
        UF : 6, UT : 5,     CONFIG: 'N U T, 0, 0, 0',
 X = -381.4 mm, Y = 572.4 mm, Z = 920.0 mm,       W = 0.0 deg, P = 0.0 deg,
    GP2:
        UF : 1, UT : 2,
       J1 = 0.0 deg, J2 = 0.0 deg
 };
P[31] {
    GP1:
        UF : 6, UT : 5,     CONFIG: 'N U T, 0, 0, 0',
       X = -389.7 mm, Y = 496.6 mm, Z = 920.0 mm,
       W = 0.0 deg, P = 0.0 deg,
    GP2:
        UF : 1, UT : 2,
       J1 = 0.0 deg, J2 = 0.0 deg
 };
P[150] {
    GP1:
        UF : 6, UT : 5,     CONFIG: 'N U T, 0, 0, 0',
 X = -372.7 mm, Y = 567.6 mm, Z = 920.0 mm,       W = 0.0 deg, P = 0.0 deg,
    GP2:
        UF : 1, UT : 2,
       J1 = 0.0 deg, J2 = 0.0 deg
 };
P[32] {
    GP1:
        UF : 6, UT : 5,     CONFIG: 'N U T, 0, 0, 0',
       X = -381.1 mm, Y = 491.6 mm, Z = 920.0 mm,
       W = 0.0 deg, P = 0.0 deg,
    GP2:
        UF : 1, UT : 2,
       J1 = 0.0 deg, J2 = 0.0 deg
 };
P[151] {
    GP1:
        UF : 6, UT : 5,     CONFIG: 'N U T, 0, 0, 0',
 X = -364.1 mm, Y = 562.6 mm, Z = 920.0 mm,       W = 0.0 deg, P = 0.0 deg,
    GP2:
        UF : 1, UT : 2,
       J1 = 0.0 deg, J2 = 0.0 deg
 };
P[33] {
    GP1:
        UF : 6, UT : 5,     CONFIG: 'N U T, 0, 0, 0',
       X = -372.5 mm, Y = 486.6 mm, Z = 920.0 mm,
       W = 0.0 deg, P = 0.0 deg,
    GP2:
        UF : 1, UT : 2,
       J1 = 0.0 deg, J2 = 0.0 deg
 };
P[152] {
    GP1:
        UF : 6, UT : 5,     CONFIG: 'N U T, 0, 0, 0',
 X = -355.5 mm, Y = 557.6 mm, Z = 920.0 mm,       W = 0.0 deg, P = 0.0 deg,
    GP2:
        UF : 1, UT : 2,
       J1 = 0.0 deg, J2 = 0.0 deg
 };
P[34] {
    GP1:
        UF : 6, UT : 5,     CONFIG: 'N U T, 0, 0, 0',
       X = -364.0 mm, Y = 481.4 mm, Z = 920.0 mm,
       W = 0.0 deg, P = 0.0 deg,
    GP2:
        UF : 1, UT : 2,
       J1 = 0.0 deg, J2 = 0.0 deg
 };
P[153] {
    GP1:
        UF : 6, UT : 5,     CONFIG: 'N U T, 0, 0, 0',
 X = -347.0 mm, Y = 552.4 mm, Z = 920.0 mm,       W = 0.0 deg, P = 0.0 deg,
    GP2:
        UF : 1, UT : 2,
       J1 = 0.0 deg, J2 = 0.0 deg
 };
P[35] {
    GP1:
        UF : 6, UT : 5,     CONFIG: 'N U T, 0, 0, 0',
       X = -355.6 mm, Y = 476.2 mm, Z = 920.0 mm,
       W = 0.0 deg, P = 0.0 deg,
    GP2:
        UF : 1, UT : 2,
       J1 = 0.0 deg, J2 = 0.0 deg
 };
P[154] {
    GP1:
        UF : 6, UT : 5,     CONFIG: 'N U T, 0, 0, 0',
 X = -338.6 mm, Y = 547.2 mm, Z = 920.0 mm,       W = 0.0 deg, P = 0.0 deg,
    GP2:
        UF : 1, UT : 2,
       J1 = 0.0 deg, J2 = 0.0 deg
 };
P[36] {
    GP1:
        UF : 6, UT : 5,     CONFIG: 'N U T, 0, 0, 0',
       X = -347.2 mm, Y = 470.8 mm, Z = 920.0 mm,
       W = 0.0 deg, P = 0.0 deg,
    GP2:
        UF : 1, UT : 2,
       J1 = 0.0 deg, J2 = 0.0 deg
 };
P[155] {
    GP1:
        UF : 6, UT : 5,     CONFIG: 'N U T, 0, 0, 0',
 X = -330.2 mm, Y = 541.8 mm, Z = 920.0 mm,       W = 0.0 deg, P = 0.0 deg,
    GP2:
        UF : 1, UT : 2,
       J1 = 0.0 deg, J2 = 0.0 deg
 };
P[37] {
    GP1:
        UF : 6, UT : 5,     CONFIG: 'N U T, 0, 0, 0',
       X = -338.9 mm, Y = 465.3 mm, Z = 920.0 mm,
       W = 0.0 deg, P = 0.0 deg,
    GP2:
        UF : 1, UT : 2,
       J1 = 0.0 deg, J2 = 0.0 deg
 };
P[156] {
    GP1:
        UF : 6, UT : 5,     CONFIG: 'N U T, 0, 0, 0',
 X = -321.9 mm, Y = 536.3 mm, Z = 920.0 mm,       W = 0.0 deg, P = 0.0 deg,
    GP2:
        UF : 1, UT : 2,
       J1 = 0.0 deg, J2 = 0.0 deg
 };
P[38] {
    GP1:
        UF : 6, UT : 5,     CONFIG: 'N U T, 0, 0, 0',
       X = -330.7 mm, Y = 459.7 mm, Z = 920.0 mm,
       W = 0.0 deg, P = 0.0 deg,
    GP2:
        UF : 1, UT : 2,
       J1 = 0.0 deg, J2 = 0.0 deg
 };
P[157] {
    GP1:
        UF : 6, UT : 5,     CONFIG: 'N U T, 0, 0, 0',
 X = -313.7 mm, Y = 530.7 mm, Z = 920.0 mm,       W = 0.0 deg, P = 0.0 deg,
    GP2:
        UF : 1, UT : 2,
       J1 = 0.0 deg, J2 = 0.0 deg
 };
P[39] {
    GP1:
        UF : 6, UT : 5,     CONFIG: 'N U T, 0, 0, 0',
       X = -322.7 mm, Y = 453.8 mm, Z = 920.0 mm,
       W = 0.0 deg, P = 0.0 deg,
    GP2:
        UF : 1, UT : 2,
       J1 = 0.0 deg, J2 = 0.0 deg
 };
P[158] {
    GP1:
        UF : 6, UT : 5,     CONFIG: 'N U T, 0, 0, 0',
 X = -305.7 mm, Y = 524.8 mm, Z = 920.0 mm,       W = 0.0 deg, P = 0.0 deg,
    GP2:
        UF : 1, UT : 2,
       J1 = 0.0 deg, J2 = 0.0 deg
 };
P[40] {
    GP1:
        UF : 6, UT : 5,     CONFIG: 'N U T, 0, 0, 0',
       X = -314.8 mm, Y = 447.8 mm, Z = 920.0 mm,
       W = 0.0 deg, P = 0.0 deg,
    GP2:
        UF : 1, UT : 2,
       J1 = 0.0 deg, J2 = 0.0 deg
 };
P[159] {
    GP1:
        UF : 6, UT : 5,     CONFIG: 'N U T, 0, 0, 0',
 X = -297.8 mm, Y = 518.8 mm, Z = 920.0 mm,       W = 0.0 deg, P = 0.0 deg,
    GP2:
        UF : 1, UT : 2,
       J1 = 0.0 deg, J2 = 0.0 deg
 };
P[41] {
    GP1:
        UF : 6, UT : 5,     CONFIG: 'N U T, 0, 0, 0',
       X = -307.1 mm, Y = 441.6 mm, Z = 920.0 mm,
       W = 0.0 deg, P = 0.0 deg,
    GP2:
        UF : 1, UT : 2,
       J1 = 0.0 deg, J2 = 0.0 deg
 };
P[160] {
    GP1:
        UF : 6, UT : 5,     CONFIG: 'N U T, 0, 0, 0',
 X = -290.1 mm, Y = 512.6 mm, Z = 920.0 mm,       W = 0.0 deg, P = 0.0 deg,
    GP2:
        UF : 1, UT : 2,
       J1 = 0.0 deg, J2 = 0.0 deg
 };
P[42] {
    GP1:
        UF : 6, UT : 5,     CONFIG: 'N U T, 0, 0, 0',
       X = -299.4 mm, Y = 435.3 mm, Z = 920.0 mm,
       W = 0.0 deg, P = 0.0 deg,
    GP2:
        UF : 1, UT : 2,
       J1 = 0.0 deg, J2 = 0.0 deg
 };
P[161] {
    GP1:
        UF : 6, UT : 5,     CONFIG: 'N U T, 0, 0, 0',
 X = -282.4 mm, Y = 506.3 mm, Z = 920.0 mm,       W = 0.0 deg, P = 0.0 deg,
    GP2:
        UF : 1, UT : 2,
       J1 = 0.0 deg, J2 = 0.0 deg
 };
P[43] {
    GP1:
        UF : 6, UT : 5,     CONFIG: 'N U T, 0, 0, 0',
       X = -291.9 mm, Y = 428.8 mm, Z = 920.0 mm,
       W = 0.0 deg, P = 0.0 deg,
    GP2:
        UF : 1, UT : 2,
       J1 = 0.0 deg, J2 = 0.0 deg
 };
P[162] {
    GP1:
        UF : 6, UT : 5,     CONFIG: 'N U T, 0, 0, 0',
 X = -274.9 mm, Y = 499.8 mm, Z = 920.0 mm,       W = 0.0 deg, P = 0.0 deg,
    GP2:
        UF : 1, UT : 2,
       J1 = 0.0 deg, J2 = 0.0 deg
 };
P[44] {
    GP1:
        UF : 6, UT : 5,     CONFIG: 'N U T, 0, 0, 0',
       X = -284.5 mm, Y = 422.2 mm, Z = 920.0 mm,
       W = 0.0 deg, P = 0.0 deg,
    GP2:
        UF : 1, UT : 2,
       J1 = 0.0 deg, J2 = 0.0 deg
 };
P[163] {
    GP1:
        UF : 6, UT : 5,     CONFIG: 'N U T, 0, 0, 0',
 X = -267.5 mm, Y = 493.2 mm, Z = 920.0 mm,       W = 0.0 deg, P = 0.0 deg,
    GP2:
        UF : 1, UT : 2,
       J1 = 0.0 deg, J2 = 0.0 deg
 };
P[45] {
    GP1:
        UF : 6, UT : 5,     CONFIG: 'N U T, 0, 0, 0',
       X = -277.2 mm, Y = 415.3 mm, Z = 920.0 mm,
       W = 0.0 deg, P = 0.0 deg,
    GP2:
        UF : 1, UT : 2,
       J1 = 0.0 deg, J2 = 0.0 deg
 };
P[164] {
    GP1:
        UF : 6, UT : 5,     CONFIG: 'N U T, 0, 0, 0',
 X = -260.2 mm, Y = 486.3 mm, Z = 920.0 mm,       W = 0.0 deg, P = 0.0 deg,
    GP2:
        UF : 1, UT : 2,
       J1 = 0.0 deg, J2 = 0.0 deg
 };
P[46] {
    GP1:
        UF : 6, UT : 5,     CONFIG: 'N U T, 0, 0, 0',
       X = -270.1 mm, Y = 408.4 mm, Z = 920.0 mm,
       W = 0.0 deg, P = 0.0 deg,
    GP2:
        UF : 1, UT : 2,
       J1 = 0.0 deg, J2 = 0.0 deg
 };
P[165] {
    GP1:
        UF : 6, UT : 5,     CONFIG: 'N U T, 0, 0, 0',
 X = -253.1 mm, Y = 479.4 mm, Z = 920.0 mm,       W = 0.0 deg, P = 0.0 deg,
    GP2:
        UF : 1, UT : 2,
       J1 = 0.0 deg, J2 = 0.0 deg
 };
P[47] {
    GP1:
        UF : 6, UT : 5,     CONFIG: 'N U T, 0, 0, 0',
       X = -263.1 mm, Y = 401.4 mm, Z = 920.0 mm,
       W = 0.0 deg, P = 0.0 deg,
    GP2:
        UF : 1, UT : 2,
       J1 = 0.0 deg, J2 = 0.0 deg
 };
P[166] {
    GP1:
        UF : 6, UT : 5,     CONFIG: 'N U T, 0, 0, 0',
 X = -246.1 mm, Y = 472.4 mm, Z = 920.0 mm,       W = 0.0 deg, P = 0.0 deg,
    GP2:
        UF : 1, UT : 2,
       J1 = 0.0 deg, J2 = 0.0 deg
 };
P[48] {
    GP1:
        UF : 6, UT : 5,     CONFIG: 'N U T, 0, 0, 0',
       X = -256.2 mm, Y = 394.2 mm, Z = 920.0 mm,
       W = 0.0 deg, P = 0.0 deg,
    GP2:
        UF : 1, UT : 2,
       J1 = 0.0 deg, J2 = 0.0 deg
 };
P[167] {
    GP1:
        UF : 6, UT : 5,     CONFIG: 'N U T, 0, 0, 0',
 X = -239.2 mm, Y = 465.2 mm, Z = 920.0 mm,       W = 0.0 deg, P = 0.0 deg,
    GP2:
        UF : 1, UT : 2,
       J1 = 0.0 deg, J2 = 0.0 deg
 };
P[49] {
    GP1:
        UF : 6, UT : 5,     CONFIG: 'N U T, 0, 0, 0',
       X = -249.5 mm, Y = 386.8 mm, Z = 920.0 mm,
       W = 0.0 deg, P = 0.0 deg,
    GP2:
        UF : 1, UT : 2,
       J1 = 0.0 deg, J2 = 0.0 deg
 };
P[168] {
    GP1:
        UF : 6, UT : 5,     CONFIG: 'N U T, 0, 0, 0',
 X = -232.5 mm, Y = 457.8 mm, Z = 920.0 mm,       W = 0.0 deg, P = 0.0 deg,
    GP2:
        UF : 1, UT : 2,
       J1 = 0.0 deg, J2 = 0.0 deg
 };
P[50] {
    GP1:
        UF : 6, UT : 5,     CONFIG: 'N U T, 0, 0, 0',
       X = -242.9 mm, Y = 379.4 mm, Z = 920.0 mm,
       W = 0.0 deg, P = 0.0 deg,
    GP2:
        UF : 1, UT : 2,
       J1 = 0.0 deg, J2 = 0.0 deg
 };
P[169] {
    GP1:
        UF : 6, UT : 5,     CONFIG: 'N U T, 0, 0, 0',
 X = -225.9 mm, Y = 450.4 mm, Z = 920.0 mm,       W = 0.0 deg, P = 0.0 deg,
    GP2:
        UF : 1, UT : 2,
       J1 = 0.0 deg, J2 = 0.0 deg
 };
P[51] {
    GP1:
        UF : 6, UT : 5,     CONFIG: 'N U T, 0, 0, 0',
       X = -236.5 mm, Y = 371.8 mm, Z = 920.0 mm,
       W = 0.0 deg, P = 0.0 deg,
    GP2:
        UF : 1, UT : 2,
       J1 = 0.0 deg, J2 = 0.0 deg
 };
P[170] {
    GP1:
        UF : 6, UT : 5,     CONFIG: 'N U T, 0, 0, 0',
 X = -219.5 mm, Y = 442.8 mm, Z = 920.0 mm,       W = 0.0 deg, P = 0.0 deg,
    GP2:
        UF : 1, UT : 2,
       J1 = 0.0 deg, J2 = 0.0 deg
 };
P[52] {
    GP1:
        UF : 6, UT : 5,     CONFIG: 'N U T, 0, 0, 0',
       X = -230.3 mm, Y = 364.1 mm, Z = 920.0 mm,
       W = 0.0 deg, P = 0.0 deg,
    GP2:
        UF : 1, UT : 2,
       J1 = 0.0 deg, J2 = 0.0 deg
 };
P[171] {
    GP1:
        UF : 6, UT : 5,     CONFIG: 'N U T, 0, 0, 0',
 X = -213.3 mm, Y = 435.1 mm, Z = 920.0 mm,       W = 0.0 deg, P = 0.0 deg,
    GP2:
        UF : 1, UT : 2,
       J1 = 0.0 deg, J2 = 0.0 deg
 };
P[53] {
    GP1:
        UF : 6, UT : 5,     CONFIG: 'N U T, 0, 0, 0',
       X = -224.2 mm, Y = 356.2 mm, Z = 920.0 mm,
       W = 0.0 deg, P = 0.0 deg,
    GP2:
        UF : 1, UT : 2,
       J1 = 0.0 deg, J2 = 0.0 deg
 };
P[172] {
    GP1:
        UF : 6, UT : 5,     CONFIG: 'N U T, 0, 0, 0',
 X = -207.2 mm, Y = 427.2 mm, Z = 920.0 mm,       W = 0.0 deg, P = 0.0 deg,
    GP2:
        UF : 1, UT : 2,
       J1 = 0.0 deg, J2 = 0.0 deg
 };
P[54] {
    GP1:
        UF : 6, UT : 5,     CONFIG: 'N U T, 0, 0, 0',
       X = -218.2 mm, Y = 348.2 mm, Z = 920.0 mm,
       W = 0.0 deg, P = 0.0 deg,
    GP2:
        UF : 1, UT : 2,
       J1 = 0.0 deg, J2 = 0.0 deg
 };
P[173] {
    GP1:
        UF : 6, UT : 5,     CONFIG: 'N U T, 0, 0, 0',
 X = -201.2 mm, Y = 419.2 mm, Z = 920.0 mm,       W = 0.0 deg, P = 0.0 deg,
    GP2:
        UF : 1, UT : 2,
       J1 = 0.0 deg, J2 = 0.0 deg
 };
P[55] {
    GP1:
        UF : 6, UT : 5,     CONFIG: 'N U T, 0, 0, 0',
       X = -212.5 mm, Y = 340.1 mm, Z = 920.0 mm,
       W = 0.0 deg, P = 0.0 deg,
    GP2:
        UF : 1, UT : 2,
       J1 = 0.0 deg, J2 = 0.0 deg
 };
P[174] {
    GP1:
        UF : 6, UT : 5,     CONFIG: 'N U T, 0, 0, 0',
 X = -195.5 mm, Y = 411.1 mm, Z = 920.0 mm,       W = 0.0 deg, P = 0.0 deg,
    GP2:
        UF : 1, UT : 2,
       J1 = 0.0 deg, J2 = 0.0 deg
 };
P[56] {
    GP1:
        UF : 6, UT : 5,     CONFIG: 'N U T, 0, 0, 0',
       X = -206.8 mm, Y = 331.9 mm, Z = 920.0 mm,
       W = 0.0 deg, P = 0.0 deg,
    GP2:
        UF : 1, UT : 2,
       J1 = 0.0 deg, J2 = 0.0 deg
 };
P[175] {
    GP1:
        UF : 6, UT : 5,     CONFIG: 'N U T, 0, 0, 0',
 X = -189.8 mm, Y = 402.9 mm, Z = 920.0 mm,       W = 0.0 deg, P = 0.0 deg,
    GP2:
        UF : 1, UT : 2,
       J1 = 0.0 deg, J2 = 0.0 deg
 };
P[57] {
    GP1:
        UF : 6, UT : 5,     CONFIG: 'N U T, 0, 0, 0',
       X = -201.4 mm, Y = 323.6 mm, Z = 920.0 mm,
       W = 0.0 deg, P = 0.0 deg,
    GP2:
        UF : 1, UT : 2,
       J1 = 0.0 deg, J2 = 0.0 deg
 };
P[176] {
    GP1:
        UF : 6, UT : 5,     CONFIG: 'N U T, 0, 0, 0',
 X = -184.4 mm, Y = 394.6 mm, Z = 920.0 mm,       W = 0.0 deg, P = 0.0 deg,
    GP2:
        UF : 1, UT : 2,
       J1 = 0.0 deg, J2 = 0.0 deg
 };
P[58] {
    GP1:
        UF : 6, UT : 5,     CONFIG: 'N U T, 0, 0, 0',
       X = -196.1 mm, Y = 315.2 mm, Z = 920.0 mm,
       W = 0.0 deg, P = 0.0 deg,
    GP2:
        UF : 1, UT : 2,
       J1 = 0.0 deg, J2 = 0.0 deg
 };
P[177] {
    GP1:
        UF : 6, UT : 5,     CONFIG: 'N U T, 0, 0, 0',
 X = -179.1 mm, Y = 386.2 mm, Z = 920.0 mm,       W = 0.0 deg, P = 0.0 deg,
    GP2:
        UF : 1, UT : 2,
       J1 = 0.0 deg, J2 = 0.0 deg
 };
P[59] {
    GP1:
        UF : 6, UT : 5,     CONFIG: 'N U T, 0, 0, 0',
       X = -190.9 mm, Y = 306.7 mm, Z = 920.0 mm,
       W = 0.0 deg, P = 0.0 deg,
    GP2:
        UF : 1, UT : 2,
       J1 = 0.0 deg, J2 = 0.0 deg
 };
P[178] {
    GP1:
        UF : 6, UT : 5,     CONFIG: 'N U T, 0, 0, 0',
 X = -173.9 mm, Y = 377.7 mm, Z = 920.0 mm,       W = 0.0 deg, P = 0.0 deg,
    GP2:
        UF : 1, UT : 2,
       J1 = 0.0 deg, J2 = 0.0 deg
 };
P[60] {
    GP1:
        UF : 6, UT : 5,     CONFIG: 'N U T, 0, 0, 0',
       X = -186.0 mm, Y = 298.1 mm, Z = 920.0 mm,
       W = 0.0 deg, P = 0.0 deg,
    GP2:
        UF : 1, UT : 2,
       J1 = 0.0 deg, J2 = 0.0 deg
 };
P[179] {
    GP1:
        UF : 6, UT : 5,     CONFIG: 'N U T, 0, 0, 0',
 X = -169.0 mm, Y = 369.1 mm, Z = 920.0 mm,       W = 0.0 deg, P = 0.0 deg,
    GP2:
        UF : 1, UT : 2,
       J1 = 0.0 deg, J2 = 0.0 deg
 };
P[61] {
    GP1:
        UF : 6, UT : 5,     CONFIG: 'N U T, 0, 0, 0',
       X = -181.1 mm, Y = 289.4 mm, Z = 920.0 mm,
       W = 0.0 deg, P = 0.0 deg,
    GP2:
        UF : 1, UT : 2,
       J1 = 0.0 deg, J2 = 0.0 deg
 };
P[180] {
    GP1:
        UF : 6, UT : 5,     CONFIG: 'N U T, 0, 0, 0',
 X = -164.1 mm, Y = 360.4 mm, Z = 920.0 mm,       W = 0.0 deg, P = 0.0 deg,
    GP2:
        UF : 1, UT : 2,
       J1 = 0.0 deg, J2 = 0.0 deg
 };
P[62] {
    GP1:
        UF : 6, UT : 5,     CONFIG: 'N U T, 0, 0, 0',
       X = -176.6 mm, Y = 280.6 mm, Z = 920.0 mm,
       W = 0.0 deg, P = 0.0 deg,
    GP2:
        UF : 1, UT : 2,
       J1 = 0.0 deg, J2 = 0.0 deg
 };
P[181] {
    GP1:
        UF : 6, UT : 5,     CONFIG: 'N U T, 0, 0, 0',
 X = -159.6 mm, Y = 351.6 mm, Z = 920.0 mm,       W = 0.0 deg, P = 0.0 deg,
    GP2:
        UF : 1, UT : 2,
       J1 = 0.0 deg, J2 = 0.0 deg
 };
P[63] {
    GP1:
        UF : 6, UT : 5,     CONFIG: 'N U T, 0, 0, 0',
       X = -172.0 mm, Y = 271.7 mm, Z = 920.0 mm,
       W = 0.0 deg, P = 0.0 deg,
    GP2:
        UF : 1, UT : 2,
       J1 = 0.0 deg, J2 = 0.0 deg
 };
P[182] {
    GP1:
        UF : 6, UT : 5,     CONFIG: 'N U T, 0, 0, 0',
 X = -155.0 mm, Y = 342.7 mm, Z = 920.0 mm,       W = 0.0 deg, P = 0.0 deg,
    GP2:
        UF : 1, UT : 2,
       J1 = 0.0 deg, J2 = 0.0 deg
 };
P[64] {
    GP1:
        UF : 6, UT : 5,     CONFIG: 'N U T, 0, 0, 0',
       X = -167.7 mm, Y = 262.7 mm, Z = 920.0 mm,
       W = 0.0 deg, P = 0.0 deg,
    GP2:
        UF : 1, UT : 2,
       J1 = 0.0 deg, J2 = 0.0 deg
 };
P[183] {
    GP1:
        UF : 6, UT : 5,     CONFIG: 'N U T, 0, 0, 0',
 X = -150.7 mm, Y = 333.7 mm, Z = 920.0 mm,       W = 0.0 deg, P = 0.0 deg,
    GP2:
        UF : 1, UT : 2,
       J1 = 0.0 deg, J2 = 0.0 deg
 };
P[65] {
    GP1:
        UF : 6, UT : 5,     CONFIG: 'N U T, 0, 0, 0',
       X = -163.5 mm, Y = 253.6 mm, Z = 920.0 mm,
       W = 0.0 deg, P = 0.0 deg,
    GP2:
        UF : 1, UT : 2,
       J1 = 0.0 deg, J2 = 0.0 deg
 };
P[184] {
    GP1:
        UF : 6, UT : 5,     CONFIG: 'N U T, 0, 0, 0',
 X = -146.5 mm, Y = 324.6 mm, Z = 920.0 mm,       W = 0.0 deg, P = 0.0 deg,
    GP2:
        UF : 1, UT : 2,
       J1 = 0.0 deg, J2 = 0.0 deg
 };
P[66] {
    GP1:
        UF : 6, UT : 5,     CONFIG: 'N U T, 0, 0, 0',
       X = -159.6 mm, Y = 244.4 mm, Z = 920.0 mm,
       W = 0.0 deg, P = 0.0 deg,
    GP2:
        UF : 1, UT : 2,
       J1 = 0.0 deg, J2 = 0.0 deg
 };
P[185] {
    GP1:
        UF : 6, UT : 5,     CONFIG: 'N U T, 0, 0, 0',
 X = -142.6 mm, Y = 315.4 mm, Z = 920.0 mm,       W = 0.0 deg, P = 0.0 deg,
    GP2:
        UF : 1, UT : 2,
       J1 = 0.0 deg, J2 = 0.0 deg
 };
P[67] {
    GP1:
        UF : 6, UT : 5,     CONFIG: 'N U T, 0, 0, 0',
       X = -155.8 mm, Y = 235.1 mm, Z = 920.0 mm,
       W = 0.0 deg, P = 0.0 deg,
    GP2:
        UF : 1, UT : 2,
       J1 = 0.0 deg, J2 = 0.0 deg
 };
P[186] {
    GP1:
        UF : 6, UT : 5,     CONFIG: 'N U T, 0, 0, 0',
 X = -138.8 mm, Y = 306.1 mm, Z = 920.0 mm,       W = 0.0 deg, P = 0.0 deg,
    GP2:
        UF : 1, UT : 2,
       J1 = 0.0 deg, J2 = 0.0 deg
 };
P[68] {
    GP1:
        UF : 6, UT : 5,     CONFIG: 'N U T, 0, 0, 0',
       X = -152.3 mm, Y = 225.8 mm, Z = 920.0 mm,
       W = 0.0 deg, P = 0.0 deg,
    GP2:
        UF : 1, UT : 2,
       J1 = 0.0 deg, J2 = 0.0 deg
 };
P[187] {
    GP1:
        UF : 6, UT : 5,     CONFIG: 'N U T, 0, 0, 0',
 X = -135.3 mm, Y = 296.8 mm, Z = 920.0 mm,       W = 0.0 deg, P = 0.0 deg,
    GP2:
        UF : 1, UT : 2,
       J1 = 0.0 deg, J2 = 0.0 deg
 };
P[69] {
    GP1:
        UF : 6, UT : 5,     CONFIG: 'N U T, 0, 0, 0',
       X = -148.9 mm, Y = 216.4 mm, Z = 920.0 mm,
       W = 0.0 deg, P = 0.0 deg,
    GP2:
        UF : 1, UT : 2,
       J1 = 0.0 deg, J2 = 0.0 deg
 };
P[188] {
    GP1:
        UF : 6, UT : 5,     CONFIG: 'N U T, 0, 0, 0',
 X = -131.9 mm, Y = 287.4 mm, Z = 920.0 mm,       W = 0.0 deg, P = 0.0 deg,
    GP2:
        UF : 1, UT : 2,
       J1 = 0.0 deg, J2 = 0.0 deg
 };
P[70] {
    GP1:
        UF : 6, UT : 5,     CONFIG: 'N U T, 0, 0, 0',
       X = -145.7 mm, Y = 206.9 mm, Z = 920.0 mm,
       W = 0.0 deg, P = 0.0 deg,
    GP2:
        UF : 1, UT : 2,
       J1 = 0.0 deg, J2 = 0.0 deg
 };
P[189] {
    GP1:
        UF : 6, UT : 5,     CONFIG: 'N U T, 0, 0, 0',
 X = -128.7 mm, Y = 277.9 mm, Z = 920.0 mm,       W = 0.0 deg, P = 0.0 deg,
    GP2:
        UF : 1, UT : 2,
       J1 = 0.0 deg, J2 = 0.0 deg
 };
P[71] {
    GP1:
        UF : 6, UT : 5,     CONFIG: 'N U T, 0, 0, 0',
       X = -142.7 mm, Y = 197.3 mm, Z = 920.0 mm,
       W = 0.0 deg, P = 0.0 deg,
    GP2:
        UF : 1, UT : 2,
       J1 = 0.0 deg, J2 = 0.0 deg
 };
P[190] {
    GP1:
        UF : 6, UT : 5,     CONFIG: 'N U T, 0, 0, 0',
 X = -125.7 mm, Y = 268.3 mm, Z = 920.0 mm,       W = 0.0 deg, P = 0.0 deg,
    GP2:
        UF : 1, UT : 2,
       J1 = 0.0 deg, J2 = 0.0 deg
 };
P[72] {
    GP1:
        UF : 6, UT : 5,     CONFIG: 'N U T, 0, 0, 0',
       X = -139.9 mm, Y = 187.7 mm, Z = 920.0 mm,
       W = 0.0 deg, P = 0.0 deg,
    GP2:
        UF : 1, UT : 2,
       J1 = 0.0 deg, J2 = 0.0 deg
 };
P[191] {
    GP1:
        UF : 6, UT : 5,     CONFIG: 'N U T, 0, 0, 0',
 X = -122.9 mm, Y = 258.7 mm, Z = 920.0 mm,       W = 0.0 deg, P = 0.0 deg,
    GP2:
        UF : 1, UT : 2,
       J1 = 0.0 deg, J2 = 0.0 deg
 };
P[73] {
    GP1:
        UF : 6, UT : 5,     CONFIG: 'N U T, 0, 0, 0',
       X = -137.2 mm, Y = 178.1 mm, Z = 920.0 mm,
       W = 0.0 deg, P = 0.0 deg,
    GP2:
        UF : 1, UT : 2,
       J1 = 0.0 deg, J2 = 0.0 deg
 };
P[192] {
    GP1:
        UF : 6, UT : 5,     CONFIG: 'N U T, 0, 0, 0',
 X = -120.2 mm, Y = 249.1 mm, Z = 920.0 mm,       W = 0.0 deg, P = 0.0 deg,
    GP2:
        UF : 1, UT : 2,
       J1 = 0.0 deg, J2 = 0.0 deg
 };
P[74] {
    GP1:
        UF : 6, UT : 5,     CONFIG: 'N U T, 0, 0, 0',
       X = -134.8 mm, Y = 168.4 mm, Z = 920.0 mm,
       W = 0.0 deg, P = 0.0 deg,
    GP2:
        UF : 1, UT : 2,
       J1 = 0.0 deg, J2 = 0.0 deg
 };
P[193] {
    GP1:
        UF : 6, UT : 5,     CONFIG: 'N U T, 0, 0, 0',
 X = -117.8 mm, Y = 239.4 mm, Z = 920.0 mm,       W = 0.0 deg, P = 0.0 deg,
    GP2:
        UF : 1, UT : 2,
       J1 = 0.0 deg, J2 = 0.0 deg
 };
P[75] {
    GP1:
        UF : 6, UT : 5,     CONFIG: 'N U T, 0, 0, 0',
       X = -132.6 mm, Y = 158.6 mm, Z = 920.0 mm,
       W = 0.0 deg, P = 0.0 deg,
    GP2:
        UF : 1, UT : 2,
       J1 = 0.0 deg, J2 = 0.0 deg
 };
P[194] {
    GP1:
        UF : 6, UT : 5,     CONFIG: 'N U T, 0, 0, 0',
 X = -115.6 mm, Y = 229.6 mm, Z = 920.0 mm,       W = 0.0 deg, P = 0.0 deg,
    GP2:
        UF : 1, UT : 2,
       J1 = 0.0 deg, J2 = 0.0 deg
 };
P[76] {
    GP1:
        UF : 6, UT : 5,     CONFIG: 'N U T, 0, 0, 0',
       X = -130.5 mm, Y = 148.9 mm, Z = 920.0 mm,
       W = 0.0 deg, P = 0.0 deg,
    GP2:
        UF : 1, UT : 2,
       J1 = 0.0 deg, J2 = 0.0 deg
 };
P[195] {
    GP1:
        UF : 6, UT : 5,     CONFIG: 'N U T, 0, 0, 0',
 X = -113.5 mm, Y = 219.9 mm, Z = 920.0 mm,       W = 0.0 deg, P = 0.0 deg,
    GP2:
        UF : 1, UT : 2,
       J1 = 0.0 deg, J2 = 0.0 deg
 };
P[77] {
    GP1:
        UF : 6, UT : 5,     CONFIG: 'N U T, 0, 0, 0',
       X = -128.7 mm, Y = 139.0 mm, Z = 920.0 mm,
       W = 0.0 deg, P = 0.0 deg,
    GP2:
        UF : 1, UT : 2,
       J1 = 0.0 deg, J2 = 0.0 deg
 };
P[196] {
    GP1:
        UF : 6, UT : 5,     CONFIG: 'N U T, 0, 0, 0',
 X = -111.7 mm, Y = 210.0 mm, Z = 920.0 mm,       W = 0.0 deg, P = 0.0 deg,
    GP2:
        UF : 1, UT : 2,
       J1 = 0.0 deg, J2 = 0.0 deg
 };
P[78] {
    GP1:
        UF : 6, UT : 5,     CONFIG: 'N U T, 0, 0, 0',
       X = -127.0 mm, Y = 129.2 mm, Z = 920.0 mm,
       W = 0.0 deg, P = 0.0 deg,
    GP2:
        UF : 1, UT : 2,
       J1 = 0.0 deg, J2 = 0.0 deg
 };
P[197] {
    GP1:
        UF : 6, UT : 5,     CONFIG: 'N U T, 0, 0, 0',
 X = -110.0 mm, Y = 200.2 mm, Z = 920.0 mm,       W = 0.0 deg, P = 0.0 deg,
    GP2:
        UF : 1, UT : 2,
       J1 = 0.0 deg, J2 = 0.0 deg
 };
P[79] {
    GP1:
        UF : 6, UT : 5,     CONFIG: 'N U T, 0, 0, 0',
       X = -125.6 mm, Y = 119.3 mm, Z = 920.0 mm,
       W = 0.0 deg, P = 0.0 deg,
    GP2:
        UF : 1, UT : 2,
       J1 = 0.0 deg, J2 = 0.0 deg
 };
P[198] {
    GP1:
        UF : 6, UT : 5,     CONFIG: 'N U T, 0, 0, 0',
 X = -108.6 mm, Y = 190.3 mm, Z = 920.0 mm,       W = 0.0 deg, P = 0.0 deg,
    GP2:
        UF : 1, UT : 2,
       J1 = 0.0 deg, J2 = 0.0 deg
 };
P[80] {
    GP1:
        UF : 6, UT : 5,     CONFIG: 'N U T, 0, 0, 0',
       X = -124.4 mm, Y = 109.4 mm, Z = 920.0 mm,
       W = 0.0 deg, P = 0.0 deg,
    GP2:
        UF : 1, UT : 2,
       J1 = 0.0 deg, J2 = 0.0 deg
 };
P[199] {
    GP1:
        UF : 6, UT : 5,     CONFIG: 'N U T, 0, 0, 0',
 X = -107.4 mm, Y = 180.4 mm, Z = 920.0 mm,       W = 0.0 deg, P = 0.0 deg,
    GP2:
        UF : 1, UT : 2,
       J1 = 0.0 deg, J2 = 0.0 deg
 };
P[81] {
    GP1:
        UF : 6, UT : 5,     CONFIG: 'N U T, 0, 0, 0',
       X = -123.4 mm, Y = 99.4 mm, Z = 920.0 mm,
       W = 0.0 deg, P = 0.0 deg,
    GP2:
        UF : 1, UT : 2,
       J1 = 0.0 deg, J2 = 0.0 deg
 };
P[200] {
    GP1:
        UF : 6, UT : 5,     CONFIG: 'N U T, 0, 0, 0',
 X = -106.4 mm, Y = 170.4 mm, Z = 920.0 mm,       W = 0.0 deg, P = 0.0 deg,
    GP2:
        UF : 1, UT : 2,
       J1 = 0.0 deg, J2 = 0.0 deg
 };
P[82] {
    GP1:
        UF : 6, UT : 5,     CONFIG: 'N U T, 0, 0, 0',
       X = -122.5 mm, Y = 89.4 mm, Z = 920.0 mm,
       W = 0.0 deg, P = 0.0 deg,
    GP2:
        UF : 1, UT : 2,
       J1 = 0.0 deg, J2 = 0.0 deg
 };
P[201] {
    GP1:
        UF : 6, UT : 5,     CONFIG: 'N U T, 0, 0, 0',
 X = -105.5 mm, Y = 160.4 mm, Z = 920.0 mm,       W = 0.0 deg, P = 0.0 deg,
    GP2:
        UF : 1, UT : 2,
       J1 = 0.0 deg, J2 = 0.0 deg
 };
P[83] {
    GP1:
        UF : 6, UT : 5,     CONFIG: 'N U T, 0, 0, 0',
       X = -121.8 mm, Y = 79.5 mm, Z = 920.0 mm,
       W = 0.0 deg, P = 0.0 deg,
    GP2:
        UF : 1, UT : 2,
       J1 = 0.0 deg, J2 = 0.0 deg
 };
P[202] {
    GP1:
        UF : 6, UT : 5,     CONFIG: 'N U T, 0, 0, 0',
 X = -104.8 mm, Y = 150.5 mm, Z = 920.0 mm,       W = 0.0 deg, P = 0.0 deg,
    GP2:
        UF : 1, UT : 2,
       J1 = 0.0 deg, J2 = 0.0 deg
 };
P[84] {
    GP1:
        UF : 6, UT : 5,     CONFIG: 'N U T, 0, 0, 0',
       X = -121.3 mm, Y = 69.5 mm, Z = 920.0 mm,
       W = 0.0 deg, P = 0.0 deg,
    GP2:
        UF : 1, UT : 2,
       J1 = 0.0 deg, J2 = 0.0 deg
 };
P[203] {
    GP1:
        UF : 6, UT : 5,     CONFIG: 'N U T, 0, 0, 0',
 X = -104.3 mm, Y = 140.5 mm, Z = 920.0 mm,       W = 0.0 deg, P = 0.0 deg,
    GP2:
        UF : 1, UT : 2,
       J1 = 0.0 deg, J2 = 0.0 deg
 };
P[85] {
    GP1:
        UF : 6, UT : 5,     CONFIG: 'N U T, 0, 0, 0',
       X = -120.8 mm, Y = 59.5 mm, Z = 920.0 mm,
       W = 0.0 deg, P = 0.0 deg,
    GP2:
        UF : 1, UT : 2,
       J1 = 0.0 deg, J2 = 0.0 deg
 };
P[204] {
    GP1:
        UF : 6, UT : 5,     CONFIG: 'N U T, 0, 0, 0',
 X = -103.8 mm, Y = 130.5 mm, Z = 920.0 mm,       W = 0.0 deg, P = 0.0 deg,
    GP2:
        UF : 1, UT : 2,
       J1 = 0.0 deg, J2 = 0.0 deg
 };
P[86] {
    GP1:
        UF : 6, UT : 5,     CONFIG: 'N U T, 0, 0, 0',
       X = -120.5 mm, Y = 49.5 mm, Z = 920.0 mm,
       W = 0.0 deg, P = 0.0 deg,
    GP2:
        UF : 1, UT : 2,
       J1 = 0.0 deg, J2 = 0.0 deg
 };
P[205] {
    GP1:
        UF : 6, UT : 5,     CONFIG: 'N U T, 0, 0, 0',
 X = -103.5 mm, Y = 120.5 mm, Z = 920.0 mm,       W = 0.0 deg, P = 0.0 deg,
    GP2:
        UF : 1, UT : 2,
       J1 = 0.0 deg, J2 = 0.0 deg
 };
P[87] {
    GP1:
        UF : 6, UT : 5,     CONFIG: 'N U T, 0, 0, 0',
       X = -120.3 mm, Y = 39.5 mm, Z = 920.0 mm,
       W = 0.0 deg, P = 0.0 deg,
    GP2:
        UF : 1, UT : 2,
       J1 = 0.0 deg, J2 = 0.0 deg
 };
P[206] {
    GP1:
        UF : 6, UT : 5,     CONFIG: 'N U T, 0, 0, 0',
 X = -103.3 mm, Y = 110.5 mm, Z = 920.0 mm,       W = 0.0 deg, P = 0.0 deg,
    GP2:
        UF : 1, UT : 2,
       J1 = 0.0 deg, J2 = 0.0 deg
 };
P[88] {
    GP1:
        UF : 6, UT : 5,     CONFIG: 'N U T, 0, 0, 0',
       X = -120.3 mm, Y = 29.5 mm, Z = 920.0 mm,
       W = 0.0 deg, P = 0.0 deg,
    GP2:
        UF : 1, UT : 2,
       J1 = 0.0 deg, J2 = 0.0 deg
 };
P[207] {
    GP1:
        UF : 6, UT : 5,     CONFIG: 'N U T, 0, 0, 0',
 X = -103.3 mm, Y = 100.5 mm, Z = 920.0 mm,       W = 0.0 deg, P = 0.0 deg,
    GP2:
        UF : 1, UT : 2,
       J1 = 0.0 deg, J2 = 0.0 deg
 };
P[89] {
    GP1:
        UF : 6, UT : 5,     CONFIG: 'N U T, 0, 0, 0',
       X = -120.5 mm, Y = 19.5 mm, Z = 920.0 mm,
       W = 0.0 deg, P = 0.0 deg,
    GP2:
        UF : 1, UT : 2,
       J1 = 0.0 deg, J2 = 0.0 deg
 };
P[208] {
    GP1:
        UF : 6, UT : 5,     CONFIG: 'N U T, 0, 0, 0',
 X = -103.5 mm, Y = 90.5 mm, Z = 920.0 mm,       W = 0.0 deg, P = 0.0 deg,
    GP2:
        UF : 1, UT : 2,
       J1 = 0.0 deg, J2 = 0.0 deg
 };
P[90] {
    GP1:
        UF : 6, UT : 5,     CONFIG: 'N U T, 0, 0, 0',
       X = -120.9 mm, Y = 9.5 mm, Z = 920.0 mm,
       W = 0.0 deg, P = 0.0 deg,
    GP2:
        UF : 1, UT : 2,
       J1 = 0.0 deg, J2 = 0.0 deg
 };
P[209] {
    GP1:
        UF : 6, UT : 5,     CONFIG: 'N U T, 0, 0, 0',
 X = -103.9 mm, Y = 80.5 mm, Z = 920.0 mm,       W = 0.0 deg, P = 0.0 deg,
    GP2:
        UF : 1, UT : 2,
       J1 = 0.0 deg, J2 = 0.0 deg
 };
P[91] {
    GP1:
        UF : 6, UT : 5,     CONFIG: 'N U T, 0, 0, 0',
       X = -121.5 mm, Y = -0.5 mm, Z = 920.0 mm,
       W = 0.0 deg, P = 0.0 deg,
    GP2:
        UF : 1, UT : 2,
       J1 = 0.0 deg, J2 = 0.0 deg
 };
P[210] {
    GP1:
        UF : 6, UT : 5,     CONFIG: 'N U T, 0, 0, 0',
 X = -104.5 mm, Y = 70.5 mm, Z = 920.0 mm,       W = 0.0 deg, P = 0.0 deg,
    GP2:
        UF : 1, UT : 2,
       J1 = 0.0 deg, J2 = 0.0 deg
 };
P[92] {
    GP1:
        UF : 6, UT : 5,     CONFIG: 'N U T, 0, 0, 0',
       X = -121.5 mm, Y = -1.7 mm, Z = 920.0 mm,
       W = 0.0 deg, P = 0.0 deg,
    GP2:
        UF : 1, UT : 2,
       J1 = 0.0 deg, J2 = 0.0 deg
 };
P[211] {
    GP1:
        UF : 6, UT : 5,     CONFIG: 'N U T, 0, 0, 0',
 X = -104.5 mm, Y = 69.3 mm, Z = 920.0 mm,       W = 0.0 deg, P = 0.0 deg,
    GP2:
        UF : 1, UT : 2,
       J1 = 0.0 deg, J2 = 0.0 deg
 };
P[93] {
    GP1:
        UF : 6, UT : 5,     CONFIG: 'N U T, 0, 0, 0',
       X = -121.4 mm, Y = -2.9 mm, Z = 920.0 mm,
       W = 0.0 deg, P = 0.0 deg,
    GP2:
        UF : 1, UT : 2,
       J1 = 0.0 deg, J2 = 0.0 deg
 };
P[212] {
    GP1:
        UF : 6, UT : 5,     CONFIG: 'N U T, 0, 0, 0',
 X = -104.4 mm, Y = 68.1 mm, Z = 920.0 mm,       W = 0.0 deg, P = 0.0 deg,
    GP2:
        UF : 1, UT : 2,
       J1 = 0.0 deg, J2 = 0.0 deg
 };
P[94] {
    GP1:
        UF : 6, UT : 5,     CONFIG: 'N U T, 0, 0, 0',
       X = -121.2 mm, Y = -4.2 mm, Z = 920.0 mm,
       W = 0.0 deg, P = 0.0 deg,
    GP2:
        UF : 1, UT : 2,
       J1 = 0.0 deg, J2 = 0.0 deg
 };
P[213] {
    GP1:
        UF : 6, UT : 5,     CONFIG: 'N U T, 0, 0, 0',
 X = -104.2 mm, Y = 66.8 mm, Z = 920.0 mm,       W = 0.0 deg, P = 0.0 deg,
    GP2:
        UF : 1, UT : 2,
       J1 = 0.0 deg, J2 = 0.0 deg
 };
P[95] {
    GP1:
        UF : 6, UT : 5,     CONFIG: 'N U T, 0, 0, 0',
       X = -120.9 mm, Y = -5.4 mm, Z = 920.0 mm,
       W = 0.0 deg, P = 0.0 deg,
    GP2:
        UF : 1, UT : 2,
       J1 = 0.0 deg, J2 = 0.0 deg
 };
P[214] {
    GP1:
        UF : 6, UT : 5,     CONFIG: 'N U T, 0, 0, 0',
 X = -103.9 mm, Y = 65.6 mm, Z = 920.0 mm,       W = 0.0 deg, P = 0.0 deg,
    GP2:
        UF : 1, UT : 2,
       J1 = 0.0 deg, J2 = 0.0 deg
 };
P[96] {
    GP1:
        UF : 6, UT : 5,     CONFIG: 'N U T, 0, 0, 0',
       X = -119.7 mm, Y = -8.3 mm, Z = 920.0 mm,
       W = 0.0 deg, P = 0.0 deg,
    GP2:
        UF : 1, UT : 2,
       J1 = 0.0 deg, J2 = 0.0 deg
 };
P[215] {
    GP1:
        UF : 6, UT : 5,     CONFIG: 'N U T, 0, 0, 0',
 X = -102.7 mm, Y = 62.7 mm, Z = 920.0 mm,       W = 0.0 deg, P = 0.0 deg,
    GP2:
        UF : 1, UT : 2,
       J1 = 0.0 deg, J2 = 0.0 deg
 };
P[97] {
    GP1:
        UF : 6, UT : 5,     CONFIG: 'N U T, 0, 0, 0',
       X = -117.9 mm, Y = -11.5 mm, Z = 920.0 mm,
       W = 0.0 deg, P = 0.0 deg,
    GP2:
        UF : 1, UT : 2,
       J1 = 0.0 deg, J2 = 0.0 deg
 };
P[216] {
    GP1:
        UF : 6, UT : 5,     CONFIG: 'N U T, 0, 0, 0',
 X = -100.9 mm, Y = 59.5 mm, Z = 920.0 mm,       W = 0.0 deg, P = 0.0 deg,
    GP2:
        UF : 1, UT : 2,
       J1 = 0.0 deg, J2 = 0.0 deg
 };
P[98] {
    GP1:
        UF : 6, UT : 5,     CONFIG: 'N U T, 0, 0, 0',
       X = -113.1 mm, Y = -20.2 mm, Z = 920.0 mm,
       W = 0.0 deg, P = 0.0 deg,
    GP2:
        UF : 1, UT : 2,
       J1 = 0.0 deg, J2 = 0.0 deg
 };
P[217] {
    GP1:
        UF : 6, UT : 5,     CONFIG: 'N U T, 0, 0, 0',
 X = -96.1 mm, Y = 50.8 mm, Z = 920.0 mm,       W = 0.0 deg, P = 0.0 deg,
    GP2:
        UF : 1, UT : 2,
       J1 = 0.0 deg, J2 = 0.0 deg
 };
P[99] {
    GP1:
        UF : 6, UT : 5,     CONFIG: 'N U T, 0, 0, 0',
       X = -108.1 mm, Y = -28.9 mm, Z = 920.0 mm,
       W = 0.0 deg, P = 0.0 deg,
    GP2:
        UF : 1, UT : 2,
       J1 = 0.0 deg, J2 = 0.0 deg
 };
P[218] {
    GP1:
        UF : 6, UT : 5,     CONFIG: 'N U T, 0, 0, 0',
 X = -91.1 mm, Y = 42.1 mm, Z = 920.0 mm,       W = 0.0 deg, P = 0.0 deg,
    GP2:
        UF : 1, UT : 2,
       J1 = 0.0 deg, J2 = 0.0 deg
 };
P[100] {
    GP1:
        UF : 6, UT : 5,     CONFIG: 'N U T, 0, 0, 0',
       X = -103.0 mm, Y = -37.5 mm, Z = 920.0 mm,
       W = 0.0 deg, P = 0.0 deg,
    GP2:
        UF : 1, UT : 2,
       J1 = 0.0 deg, J2 = 0.0 deg
 };
P[219] {
    GP1:
        UF : 6, UT : 5,     CONFIG: 'N U T, 0, 0, 0',
 X = -86.0 mm, Y = 33.5 mm, Z = 920.0 mm,       W = 0.0 deg, P = 0.0 deg,
    GP2:
        UF : 1, UT : 2,
       J1 = 0.0 deg, J2 = 0.0 deg
 };
P[101] {
    GP1:
        UF : 6, UT : 5,     CONFIG: 'N U T, 0, 0, 0',
       X = -101.7 mm, Y = -39.0 mm, Z = 920.0 mm,
       W = 0.0 deg, P = 0.0 deg,
    GP2:
        UF : 1, UT : 2,
       J1 = 0.0 deg, J2 = 0.0 deg
 };
P[220] {
    GP1:
        UF : 6, UT : 5,     CONFIG: 'N U T, 0, 0, 0',
 X = -84.7 mm, Y = 32.0 mm, Z = 920.0 mm,       W = 0.0 deg, P = 0.0 deg,
    GP2:
        UF : 1, UT : 2,
       J1 = 0.0 deg, J2 = 0.0 deg
 };
P[102] {
    GP1:
        UF : 6, UT : 5,     CONFIG: 'N U T, 0, 0, 0',
       X = -100.4 mm, Y = -39.8 mm, Z = 920.0 mm,
       W = 0.0 deg, P = 0.0 deg,
    GP2:
        UF : 1, UT : 2,
       J1 = 0.0 deg, J2 = 0.0 deg
 };
P[221] {
    GP1:
        UF : 6, UT : 5,     CONFIG: 'N U T, 0, 0, 0',
 X = -83.4 mm, Y = 31.2 mm, Z = 920.0 mm,       W = 0.0 deg, P = 0.0 deg,
    GP2:
        UF : 1, UT : 2,
       J1 = 0.0 deg, J2 = 0.0 deg
 };
P[103] {
    GP1:
        UF : 6, UT : 5,     CONFIG: 'N U T, 0, 0, 0',
       X = -99.0 mm, Y = -40.5 mm, Z = 920.0 mm,
       W = 0.0 deg, P = 0.0 deg,
    GP2:
        UF : 1, UT : 2,
       J1 = 0.0 deg, J2 = 0.0 deg
 };
P[222] {
    GP1:
        UF : 6, UT : 5,     CONFIG: 'N U T, 0, 0, 0',
 X = -82.0 mm, Y = 30.5 mm, Z = 920.0 mm,       W = 0.0 deg, P = 0.0 deg,
    GP2:
        UF : 1, UT : 2,
       J1 = 0.0 deg, J2 = 0.0 deg
 };
P[104] {
    GP1:
        UF : 6, UT : 5,     CONFIG: 'N U T, 0, 0, 0',
       X = -97.3 mm, Y = -40.8 mm, Z = 920.0 mm,
       W = 0.0 deg, P = 0.0 deg,
    GP2:
        UF : 1, UT : 2,
       J1 = 0.0 deg, J2 = 0.0 deg
 };
P[223] {
    GP1:
        UF : 6, UT : 5,     CONFIG: 'N U T, 0, 0, 0',
 X = -80.3 mm, Y = 30.2 mm, Z = 920.0 mm,       W = 0.0 deg, P = 0.0 deg,
    GP2:
        UF : 1, UT : 2,
       J1 = 0.0 deg, J2 = 0.0 deg
 };
P[105] {
    GP1:
        UF : 6, UT : 5,     CONFIG: 'N U T, 0, 0, 0',
       X = -95.6 mm, Y = -40.8 mm, Z = 920.0 mm,
       W = 0.0 deg, P = 0.0 deg,
    GP2:
        UF : 1, UT : 2,
       J1 = 0.0 deg, J2 = 0.0 deg
 };
P[224] {
    GP1:
        UF : 6, UT : 5,     CONFIG: 'N U T, 0, 0, 0',
 X = -78.6 mm, Y = 30.2 mm, Z = 920.0 mm,       W = 0.0 deg, P = 0.0 deg,
    GP2:
        UF : 1, UT : 2,
       J1 = 0.0 deg, J2 = 0.0 deg
 };
P[106] {
    GP1:
        UF : 6, UT : 5,     CONFIG: 'N U T, 0, 0, 0',
       X = -94.0 mm, Y = -40.4 mm, Z = 920.0 mm,
       W = 0.0 deg, P = 0.0 deg,
    GP2:
        UF : 1, UT : 2,
       J1 = 0.0 deg, J2 = 0.0 deg
 };
P[225] {
    GP1:
        UF : 6, UT : 5,     CONFIG: 'N U T, 0, 0, 0',
 X = -77.0 mm, Y = 30.6 mm, Z = 920.0 mm,       W = 0.0 deg, P = 0.0 deg,
    GP2:
        UF : 1, UT : 2,
       J1 = 0.0 deg, J2 = 0.0 deg
 };
P[107] {
    GP1:
        UF : 6, UT : 5,     CONFIG: 'N U T, 0, 0, 0',
       X = -92.5 mm, Y = -39.8 mm, Z = 920.0 mm,
       W = 0.0 deg, P = 0.0 deg,
    GP2:
        UF : 1, UT : 2,
       J1 = 0.0 deg, J2 = 0.0 deg
 };
P[226] {
    GP1:
        UF : 6, UT : 5,     CONFIG: 'N U T, 0, 0, 0',
 X = -75.5 mm, Y = 31.2 mm, Z = 920.0 mm,       W = 0.0 deg, P = 0.0 deg,
    GP2:
        UF : 1, UT : 2,
       J1 = 0.0 deg, J2 = 0.0 deg
 };
P[108] {
    GP1:
        UF : 6, UT : 5,     CONFIG: 'N U T, 0, 0, 0',
       X = -90.9 mm, Y = -39.0 mm, Z = 920.0 mm,
       W = 0.0 deg, P = 0.0 deg,
    GP2:
        UF : 1, UT : 2,
       J1 = 0.0 deg, J2 = 0.0 deg
 };
P[227] {
    GP1:
        UF : 6, UT : 5,     CONFIG: 'N U T, 0, 0, 0',
 X = -73.9 mm, Y = 32.0 mm, Z = 920.0 mm,       W = 0.0 deg, P = 0.0 deg,
    GP2:
        UF : 1, UT : 2,
       J1 = 0.0 deg, J2 = 0.0 deg
 };
P[109] {
    GP1:
        UF : 6, UT : 5,     CONFIG: 'N U T, 0, 0, 0',
       X = -87.3 mm, Y = -36.9 mm, Z = 920.0 mm,
       W = 0.0 deg, P = 0.0 deg,
    GP2:
        UF : 1, UT : 2,
       J1 = 0.0 deg, J2 = 0.0 deg
 };
P[228] {
    GP1:
        UF : 6, UT : 5,     CONFIG: 'N U T, 0, 0, 0',
 X = -70.3 mm, Y = 34.1 mm, Z = 920.0 mm,       W = 0.0 deg, P = 0.0 deg,
    GP2:
        UF : 1, UT : 2,
       J1 = 0.0 deg, J2 = 0.0 deg
 };
P[110] {
    GP1:
        UF : 6, UT : 5,     CONFIG: 'N U T, 0, 0, 0',
       X = -78.5 mm, Y = -32.1 mm, Z = 920.0 mm,
       W = 0.0 deg, P = 0.0 deg,
    GP2:
        UF : 1, UT : 2,
       J1 = 0.0 deg, J2 = 0.0 deg
 };
P[229] {
    GP1:
        UF : 6, UT : 5,     CONFIG: 'N U T, 0, 0, 0',
 X = -61.5 mm, Y = 38.9 mm, Z = 920.0 mm,       W = 0.0 deg, P = 0.0 deg,
    GP2:
        UF : 1, UT : 2,
       J1 = 0.0 deg, J2 = 0.0 deg
 };
P[111] {
    GP1:
        UF : 6, UT : 5,     CONFIG: 'N U T, 0, 0, 0',
       X = -69.8 mm, Y = -27.2 mm, Z = 920.0 mm,
       W = 0.0 deg, P = 0.0 deg,
    GP2:
        UF : 1, UT : 2,
       J1 = 0.0 deg, J2 = 0.0 deg
 };
P[230] {
    GP1:
        UF : 6, UT : 5,     CONFIG: 'N U T, 0, 0, 0',
 X = -52.8 mm, Y = 43.8 mm, Z = 920.0 mm,       W = 0.0 deg, P = 0.0 deg,
    GP2:
        UF : 1, UT : 2,
       J1 = 0.0 deg, J2 = 0.0 deg
 };
P[112] {
    GP1:
        UF : 6, UT : 5,     CONFIG: 'N U T, 0, 0, 0',
       X = -61.0 mm, Y = -22.4 mm, Z = 920.0 mm,
       W = 0.0 deg, P = 0.0 deg,
    GP2:
        UF : 1, UT : 2,
       J1 = 0.0 deg, J2 = 0.0 deg
 };
P[231] {
    GP1:
        UF : 6, UT : 5,     CONFIG: 'N U T, 0, 0, 0',
 X = -44.0 mm, Y = 48.6 mm, Z = 920.0 mm,       W = 0.0 deg, P = 0.0 deg,
    GP2:
        UF : 1, UT : 2,
       J1 = 0.0 deg, J2 = 0.0 deg
 };
P[113] {
    GP1:
        UF : 6, UT : 5,     CONFIG: 'N U T, 0, 0, 0',
       X = -52.3 mm, Y = -17.6 mm, Z = 920.0 mm,
       W = 0.0 deg, P = 0.0 deg,
    GP2:
        UF : 1, UT : 2,
       J1 = 0.0 deg, J2 = 0.0 deg
 };
P[232] {
    GP1:
        UF : 6, UT : 5,     CONFIG: 'N U T, 0, 0, 0',
 X = -35.3 mm, Y = 53.4 mm, Z = 920.0 mm,       W = 0.0 deg, P = 0.0 deg,
    GP2:
        UF : 1, UT : 2,
       J1 = 0.0 deg, J2 = 0.0 deg
 };
P[114] {
    GP1:
        UF : 6, UT : 5,     CONFIG: 'N U T, 0, 0, 0',
       X = -43.6 mm, Y = -12.7 mm, Z = 920.0 mm,
       W = 0.0 deg, P = 0.0 deg,
    GP2:
        UF : 1, UT : 2,
       J1 = 0.0 deg, J2 = 0.0 deg
 };
P[233] {
    GP1:
        UF : 6, UT : 5,     CONFIG: 'N U T, 0, 0, 0',
 X = -26.6 mm, Y = 58.3 mm, Z = 920.0 mm,       W = 0.0 deg, P = 0.0 deg,
    GP2:
        UF : 1, UT : 2,
       J1 = 0.0 deg, J2 = 0.0 deg
 };
P[115] {
    GP1:
        UF : 6, UT : 5,     CONFIG: 'N U T, 0, 0, 0',
       X = -34.8 mm, Y = -7.9 mm, Z = 920.0 mm,
       W = 0.0 deg, P = 0.0 deg,
    GP2:
        UF : 1, UT : 2,
       J1 = 0.0 deg, J2 = 0.0 deg
 };
P[234] {
    GP1:
        UF : 6, UT : 5,     CONFIG: 'N U T, 0, 0, 0',
 X = -17.8 mm, Y = 63.1 mm, Z = 920.0 mm,       W = 0.0 deg, P = 0.0 deg,
    GP2:
        UF : 1, UT : 2,
       J1 = 0.0 deg, J2 = 0.0 deg
 };
P[116] {
    GP1:
        UF : 6, UT : 5,     CONFIG: 'N U T, 0, 0, 0',
       X = -26.1 mm, Y = -3.0 mm, Z = 920.0 mm,
       W = 0.0 deg, P = 0.0 deg,
    GP2:
        UF : 1, UT : 2,
       J1 = 0.0 deg, J2 = 0.0 deg
 };
P[235] {
    GP1:
        UF : 6, UT : 5,     CONFIG: 'N U T, 0, 0, 0',
 X = -9.1 mm, Y = 68.0 mm, Z = 920.0 mm,       W = 0.0 deg, P = 0.0 deg,
    GP2:
        UF : 1, UT : 2,
       J1 = 0.0 deg, J2 = 0.0 deg
 };
P[117] {
    GP1:
        UF : 6, UT : 5,     CONFIG: 'N U T, 0, 0, 0',
       X = -17.3 mm, Y = 1.8 mm, Z = 920.0 mm,
       W = 0.0 deg, P = 0.0 deg,
    GP2:
        UF : 1, UT : 2,
       J1 = 0.0 deg, J2 = 0.0 deg
 };
P[236] {
    GP1:
        UF : 6, UT : 5,     CONFIG: 'N U T, 0, 0, 0',
 X = -0.3 mm, Y = 72.8 mm, Z = 920.0 mm,       W = 0.0 deg, P = 0.0 deg,
    GP2:
        UF : 1, UT : 2,
       J1 = 0.0 deg, J2 = 0.0 deg
 };
/END
